IF SUPER^.Step(881, TRUE, 'Step number 881') THEN
    SUPER^.StepCompleteWhen((_runOneStep OR _runAllSteps) AND _finishStep);

    IF _runOneStep THEN
        _runOneStep := FALSE;
        RETURN;
    END_IF
END_IF

IF SUPER^.Step(882, TRUE, 'Step number 882') THEN
    SUPER^.StepCompleteWhen((_runOneStep OR _runAllSteps) AND _finishStep);

    IF _runOneStep THEN
        _runOneStep := FALSE;
        RETURN;
    END_IF
END_IF

IF SUPER^.Step(883, TRUE, 'Step number 883') THEN
    SUPER^.StepCompleteWhen((_runOneStep OR _runAllSteps) AND _finishStep);

    IF _runOneStep THEN
        _runOneStep := FALSE;
        RETURN;
    END_IF
END_IF

IF SUPER^.Step(884, TRUE, 'Step number 884') THEN
    SUPER^.StepCompleteWhen((_runOneStep OR _runAllSteps) AND _finishStep);

    IF _runOneStep THEN
        _runOneStep := FALSE;
        RETURN;
    END_IF
END_IF

IF SUPER^.Step(885, TRUE, 'Step number 885') THEN
    SUPER^.StepCompleteWhen((_runOneStep OR _runAllSteps) AND _finishStep);

    IF _runOneStep THEN
        _runOneStep := FALSE;
        RETURN;
    END_IF
END_IF

IF SUPER^.Step(886, TRUE, 'Step number 886') THEN
    SUPER^.StepCompleteWhen((_runOneStep OR _runAllSteps) AND _finishStep);

    IF _runOneStep THEN
        _runOneStep := FALSE;
        RETURN;
    END_IF
END_IF

IF SUPER^.Step(887, TRUE, 'Step number 887') THEN
    SUPER^.StepCompleteWhen((_runOneStep OR _runAllSteps) AND _finishStep);

    IF _runOneStep THEN
        _runOneStep := FALSE;
        RETURN;
    END_IF
END_IF

IF SUPER^.Step(888, TRUE, 'Step number 888') THEN
    SUPER^.StepCompleteWhen((_runOneStep OR _runAllSteps) AND _finishStep);

    IF _runOneStep THEN
        _runOneStep := FALSE;
        RETURN;
    END_IF
END_IF

IF SUPER^.Step(889, TRUE, 'Step number 889') THEN
    SUPER^.StepCompleteWhen((_runOneStep OR _runAllSteps) AND _finishStep);

    IF _runOneStep THEN
        _runOneStep := FALSE;
        RETURN;
    END_IF
END_IF

IF SUPER^.Step(890, TRUE, 'Step number 890') THEN
    SUPER^.StepCompleteWhen((_runOneStep OR _runAllSteps) AND _finishStep);

    IF _runOneStep THEN
        _runOneStep := FALSE;
        RETURN;
    END_IF
END_IF

IF SUPER^.Step(891, TRUE, 'Step number 891') THEN
    SUPER^.StepCompleteWhen((_runOneStep OR _runAllSteps) AND _finishStep);

    IF _runOneStep THEN
        _runOneStep := FALSE;
        RETURN;
    END_IF
END_IF

IF SUPER^.Step(892, TRUE, 'Step number 892') THEN
    SUPER^.StepCompleteWhen((_runOneStep OR _runAllSteps) AND _finishStep);

    IF _runOneStep THEN
        _runOneStep := FALSE;
        RETURN;
    END_IF
END_IF

IF SUPER^.Step(893, TRUE, 'Step number 893') THEN
    SUPER^.StepCompleteWhen((_runOneStep OR _runAllSteps) AND _finishStep);

    IF _runOneStep THEN
        _runOneStep := FALSE;
        RETURN;
    END_IF
END_IF

IF SUPER^.Step(894, TRUE, 'Step number 894') THEN
    SUPER^.StepCompleteWhen((_runOneStep OR _runAllSteps) AND _finishStep);

    IF _runOneStep THEN
        _runOneStep := FALSE;
        RETURN;
    END_IF
END_IF

IF SUPER^.Step(895, TRUE, 'Step number 895') THEN
    SUPER^.StepCompleteWhen((_runOneStep OR _runAllSteps) AND _finishStep);

    IF _runOneStep THEN
        _runOneStep := FALSE;
        RETURN;
    END_IF
END_IF

IF SUPER^.Step(896, TRUE, 'Step number 896') THEN
    SUPER^.StepCompleteWhen((_runOneStep OR _runAllSteps) AND _finishStep);

    IF _runOneStep THEN
        _runOneStep := FALSE;
        RETURN;
    END_IF
END_IF

IF SUPER^.Step(897, TRUE, 'Step number 897') THEN
    SUPER^.StepCompleteWhen((_runOneStep OR _runAllSteps) AND _finishStep);

    IF _runOneStep THEN
        _runOneStep := FALSE;
        RETURN;
    END_IF
END_IF

IF SUPER^.Step(898, TRUE, 'Step number 898') THEN
    SUPER^.StepCompleteWhen((_runOneStep OR _runAllSteps) AND _finishStep);

    IF _runOneStep THEN
        _runOneStep := FALSE;
        RETURN;
    END_IF
END_IF

IF SUPER^.Step(899, TRUE, 'Step number 899') THEN
    SUPER^.StepCompleteWhen((_runOneStep OR _runAllSteps) AND _finishStep);

    IF _runOneStep THEN
        _runOneStep := FALSE;
        RETURN;
    END_IF
END_IF

IF SUPER^.Step(900, TRUE, 'Step number 900') THEN
    SUPER^.StepCompleteWhen((_runOneStep OR _runAllSteps) AND _finishStep);

    IF _runOneStep THEN
        _runOneStep := FALSE;
        RETURN;
    END_IF
END_IF

IF SUPER^.Step(901, TRUE, 'Step number 901') THEN
    SUPER^.StepCompleteWhen((_runOneStep OR _runAllSteps) AND _finishStep);

    IF _runOneStep THEN
        _runOneStep := FALSE;
        RETURN;
    END_IF
END_IF

IF SUPER^.Step(902, TRUE, 'Step number 902') THEN
    SUPER^.StepCompleteWhen((_runOneStep OR _runAllSteps) AND _finishStep);

    IF _runOneStep THEN
        _runOneStep := FALSE;
        RETURN;
    END_IF
END_IF

IF SUPER^.Step(903, TRUE, 'Step number 903') THEN
    SUPER^.StepCompleteWhen((_runOneStep OR _runAllSteps) AND _finishStep);

    IF _runOneStep THEN
        _runOneStep := FALSE;
        RETURN;
    END_IF
END_IF

IF SUPER^.Step(904, TRUE, 'Step number 904') THEN
    SUPER^.StepCompleteWhen((_runOneStep OR _runAllSteps) AND _finishStep);

    IF _runOneStep THEN
        _runOneStep := FALSE;
        RETURN;
    END_IF
END_IF

IF SUPER^.Step(905, TRUE, 'Step number 905') THEN
    SUPER^.StepCompleteWhen((_runOneStep OR _runAllSteps) AND _finishStep);

    IF _runOneStep THEN
        _runOneStep := FALSE;
        RETURN;
    END_IF
END_IF

IF SUPER^.Step(906, TRUE, 'Step number 906') THEN
    SUPER^.StepCompleteWhen((_runOneStep OR _runAllSteps) AND _finishStep);

    IF _runOneStep THEN
        _runOneStep := FALSE;
        RETURN;
    END_IF
END_IF

IF SUPER^.Step(907, TRUE, 'Step number 907') THEN
    SUPER^.StepCompleteWhen((_runOneStep OR _runAllSteps) AND _finishStep);

    IF _runOneStep THEN
        _runOneStep := FALSE;
        RETURN;
    END_IF
END_IF

IF SUPER^.Step(908, TRUE, 'Step number 908') THEN
    SUPER^.StepCompleteWhen((_runOneStep OR _runAllSteps) AND _finishStep);

    IF _runOneStep THEN
        _runOneStep := FALSE;
        RETURN;
    END_IF
END_IF

IF SUPER^.Step(909, TRUE, 'Step number 909') THEN
    SUPER^.StepCompleteWhen((_runOneStep OR _runAllSteps) AND _finishStep);

    IF _runOneStep THEN
        _runOneStep := FALSE;
        RETURN;
    END_IF
END_IF

IF SUPER^.Step(910, TRUE, 'Step number 910') THEN
    SUPER^.StepCompleteWhen((_runOneStep OR _runAllSteps) AND _finishStep);

    IF _runOneStep THEN
        _runOneStep := FALSE;
        RETURN;
    END_IF
END_IF

IF SUPER^.Step(911, TRUE, 'Step number 911') THEN
    SUPER^.StepCompleteWhen((_runOneStep OR _runAllSteps) AND _finishStep);

    IF _runOneStep THEN
        _runOneStep := FALSE;
        RETURN;
    END_IF
END_IF

IF SUPER^.Step(912, TRUE, 'Step number 912') THEN
    SUPER^.StepCompleteWhen((_runOneStep OR _runAllSteps) AND _finishStep);

    IF _runOneStep THEN
        _runOneStep := FALSE;
        RETURN;
    END_IF
END_IF

IF SUPER^.Step(913, TRUE, 'Step number 913') THEN
    SUPER^.StepCompleteWhen((_runOneStep OR _runAllSteps) AND _finishStep);

    IF _runOneStep THEN
        _runOneStep := FALSE;
        RETURN;
    END_IF
END_IF

IF SUPER^.Step(914, TRUE, 'Step number 914') THEN
    SUPER^.StepCompleteWhen((_runOneStep OR _runAllSteps) AND _finishStep);

    IF _runOneStep THEN
        _runOneStep := FALSE;
        RETURN;
    END_IF
END_IF

IF SUPER^.Step(915, TRUE, 'Step number 915') THEN
    SUPER^.StepCompleteWhen((_runOneStep OR _runAllSteps) AND _finishStep);

    IF _runOneStep THEN
        _runOneStep := FALSE;
        RETURN;
    END_IF
END_IF

IF SUPER^.Step(916, TRUE, 'Step number 916') THEN
    SUPER^.StepCompleteWhen((_runOneStep OR _runAllSteps) AND _finishStep);

    IF _runOneStep THEN
        _runOneStep := FALSE;
        RETURN;
    END_IF
END_IF

IF SUPER^.Step(917, TRUE, 'Step number 917') THEN
    SUPER^.StepCompleteWhen((_runOneStep OR _runAllSteps) AND _finishStep);

    IF _runOneStep THEN
        _runOneStep := FALSE;
        RETURN;
    END_IF
END_IF

IF SUPER^.Step(918, TRUE, 'Step number 918') THEN
    SUPER^.StepCompleteWhen((_runOneStep OR _runAllSteps) AND _finishStep);

    IF _runOneStep THEN
        _runOneStep := FALSE;
        RETURN;
    END_IF
END_IF

IF SUPER^.Step(919, TRUE, 'Step number 919') THEN
    SUPER^.StepCompleteWhen((_runOneStep OR _runAllSteps) AND _finishStep);

    IF _runOneStep THEN
        _runOneStep := FALSE;
        RETURN;
    END_IF
END_IF

IF SUPER^.Step(920, TRUE, 'Step number 920') THEN
    SUPER^.StepCompleteWhen((_runOneStep OR _runAllSteps) AND _finishStep);

    IF _runOneStep THEN
        _runOneStep := FALSE;
        RETURN;
    END_IF
END_IF

IF SUPER^.Step(921, TRUE, 'Step number 921') THEN
    SUPER^.StepCompleteWhen((_runOneStep OR _runAllSteps) AND _finishStep);

    IF _runOneStep THEN
        _runOneStep := FALSE;
        RETURN;
    END_IF
END_IF

IF SUPER^.Step(922, TRUE, 'Step number 922') THEN
    SUPER^.StepCompleteWhen((_runOneStep OR _runAllSteps) AND _finishStep);

    IF _runOneStep THEN
        _runOneStep := FALSE;
        RETURN;
    END_IF
END_IF

IF SUPER^.Step(923, TRUE, 'Step number 923') THEN
    SUPER^.StepCompleteWhen((_runOneStep OR _runAllSteps) AND _finishStep);

    IF _runOneStep THEN
        _runOneStep := FALSE;
        RETURN;
    END_IF
END_IF

IF SUPER^.Step(924, TRUE, 'Step number 924') THEN
    SUPER^.StepCompleteWhen((_runOneStep OR _runAllSteps) AND _finishStep);

    IF _runOneStep THEN
        _runOneStep := FALSE;
        RETURN;
    END_IF
END_IF

IF SUPER^.Step(925, TRUE, 'Step number 925') THEN
    SUPER^.StepCompleteWhen((_runOneStep OR _runAllSteps) AND _finishStep);

    IF _runOneStep THEN
        _runOneStep := FALSE;
        RETURN;
    END_IF
END_IF

IF SUPER^.Step(926, TRUE, 'Step number 926') THEN
    SUPER^.StepCompleteWhen((_runOneStep OR _runAllSteps) AND _finishStep);

    IF _runOneStep THEN
        _runOneStep := FALSE;
        RETURN;
    END_IF
END_IF

IF SUPER^.Step(927, TRUE, 'Step number 927') THEN
    SUPER^.StepCompleteWhen((_runOneStep OR _runAllSteps) AND _finishStep);

    IF _runOneStep THEN
        _runOneStep := FALSE;
        RETURN;
    END_IF
END_IF

IF SUPER^.Step(928, TRUE, 'Step number 928') THEN
    SUPER^.StepCompleteWhen((_runOneStep OR _runAllSteps) AND _finishStep);

    IF _runOneStep THEN
        _runOneStep := FALSE;
        RETURN;
    END_IF
END_IF

IF SUPER^.Step(929, TRUE, 'Step number 929') THEN
    SUPER^.StepCompleteWhen((_runOneStep OR _runAllSteps) AND _finishStep);

    IF _runOneStep THEN
        _runOneStep := FALSE;
        RETURN;
    END_IF
END_IF

IF SUPER^.Step(930, TRUE, 'Step number 930') THEN
    SUPER^.StepCompleteWhen((_runOneStep OR _runAllSteps) AND _finishStep);

    IF _runOneStep THEN
        _runOneStep := FALSE;
        RETURN;
    END_IF
END_IF

IF SUPER^.Step(931, TRUE, 'Step number 931') THEN
    SUPER^.StepCompleteWhen((_runOneStep OR _runAllSteps) AND _finishStep);

    IF _runOneStep THEN
        _runOneStep := FALSE;
        RETURN;
    END_IF
END_IF

IF SUPER^.Step(932, TRUE, 'Step number 932') THEN
    SUPER^.StepCompleteWhen((_runOneStep OR _runAllSteps) AND _finishStep);

    IF _runOneStep THEN
        _runOneStep := FALSE;
        RETURN;
    END_IF
END_IF

IF SUPER^.Step(933, TRUE, 'Step number 933') THEN
    SUPER^.StepCompleteWhen((_runOneStep OR _runAllSteps) AND _finishStep);

    IF _runOneStep THEN
        _runOneStep := FALSE;
        RETURN;
    END_IF
END_IF

IF SUPER^.Step(934, TRUE, 'Step number 934') THEN
    SUPER^.StepCompleteWhen((_runOneStep OR _runAllSteps) AND _finishStep);

    IF _runOneStep THEN
        _runOneStep := FALSE;
        RETURN;
    END_IF
END_IF

IF SUPER^.Step(935, TRUE, 'Step number 935') THEN
    SUPER^.StepCompleteWhen((_runOneStep OR _runAllSteps) AND _finishStep);

    IF _runOneStep THEN
        _runOneStep := FALSE;
        RETURN;
    END_IF
END_IF

IF SUPER^.Step(936, TRUE, 'Step number 936') THEN
    SUPER^.StepCompleteWhen((_runOneStep OR _runAllSteps) AND _finishStep);

    IF _runOneStep THEN
        _runOneStep := FALSE;
        RETURN;
    END_IF
END_IF

IF SUPER^.Step(937, TRUE, 'Step number 937') THEN
    SUPER^.StepCompleteWhen((_runOneStep OR _runAllSteps) AND _finishStep);

    IF _runOneStep THEN
        _runOneStep := FALSE;
        RETURN;
    END_IF
END_IF

IF SUPER^.Step(938, TRUE, 'Step number 938') THEN
    SUPER^.StepCompleteWhen((_runOneStep OR _runAllSteps) AND _finishStep);

    IF _runOneStep THEN
        _runOneStep := FALSE;
        RETURN;
    END_IF
END_IF

IF SUPER^.Step(939, TRUE, 'Step number 939') THEN
    SUPER^.StepCompleteWhen((_runOneStep OR _runAllSteps) AND _finishStep);

    IF _runOneStep THEN
        _runOneStep := FALSE;
        RETURN;
    END_IF
END_IF

IF SUPER^.Step(940, TRUE, 'Step number 940') THEN
    SUPER^.StepCompleteWhen((_runOneStep OR _runAllSteps) AND _finishStep);

    IF _runOneStep THEN
        _runOneStep := FALSE;
        RETURN;
    END_IF
END_IF

IF SUPER^.Step(941, TRUE, 'Step number 941') THEN
    SUPER^.StepCompleteWhen((_runOneStep OR _runAllSteps) AND _finishStep);

    IF _runOneStep THEN
        _runOneStep := FALSE;
        RETURN;
    END_IF
END_IF

IF SUPER^.Step(942, TRUE, 'Step number 942') THEN
    SUPER^.StepCompleteWhen((_runOneStep OR _runAllSteps) AND _finishStep);

    IF _runOneStep THEN
        _runOneStep := FALSE;
        RETURN;
    END_IF
END_IF

IF SUPER^.Step(943, TRUE, 'Step number 943') THEN
    SUPER^.StepCompleteWhen((_runOneStep OR _runAllSteps) AND _finishStep);

    IF _runOneStep THEN
        _runOneStep := FALSE;
        RETURN;
    END_IF
END_IF

IF SUPER^.Step(944, TRUE, 'Step number 944') THEN
    SUPER^.StepCompleteWhen((_runOneStep OR _runAllSteps) AND _finishStep);

    IF _runOneStep THEN
        _runOneStep := FALSE;
        RETURN;
    END_IF
END_IF

IF SUPER^.Step(945, TRUE, 'Step number 945') THEN
    SUPER^.StepCompleteWhen((_runOneStep OR _runAllSteps) AND _finishStep);

    IF _runOneStep THEN
        _runOneStep := FALSE;
        RETURN;
    END_IF
END_IF

IF SUPER^.Step(946, TRUE, 'Step number 946') THEN
    SUPER^.StepCompleteWhen((_runOneStep OR _runAllSteps) AND _finishStep);

    IF _runOneStep THEN
        _runOneStep := FALSE;
        RETURN;
    END_IF
END_IF

IF SUPER^.Step(947, TRUE, 'Step number 947') THEN
    SUPER^.StepCompleteWhen((_runOneStep OR _runAllSteps) AND _finishStep);

    IF _runOneStep THEN
        _runOneStep := FALSE;
        RETURN;
    END_IF
END_IF

IF SUPER^.Step(948, TRUE, 'Step number 948') THEN
    SUPER^.StepCompleteWhen((_runOneStep OR _runAllSteps) AND _finishStep);

    IF _runOneStep THEN
        _runOneStep := FALSE;
        RETURN;
    END_IF
END_IF

IF SUPER^.Step(949, TRUE, 'Step number 949') THEN
    SUPER^.StepCompleteWhen((_runOneStep OR _runAllSteps) AND _finishStep);

    IF _runOneStep THEN
        _runOneStep := FALSE;
        RETURN;
    END_IF
END_IF

IF SUPER^.Step(950, TRUE, 'Step number 950') THEN
    SUPER^.StepCompleteWhen((_runOneStep OR _runAllSteps) AND _finishStep);

    IF _runOneStep THEN
        _runOneStep := FALSE;
        RETURN;
    END_IF
END_IF

IF SUPER^.Step(951, TRUE, 'Step number 951') THEN
    SUPER^.StepCompleteWhen((_runOneStep OR _runAllSteps) AND _finishStep);

    IF _runOneStep THEN
        _runOneStep := FALSE;
        RETURN;
    END_IF
END_IF

IF SUPER^.Step(952, TRUE, 'Step number 952') THEN
    SUPER^.StepCompleteWhen((_runOneStep OR _runAllSteps) AND _finishStep);

    IF _runOneStep THEN
        _runOneStep := FALSE;
        RETURN;
    END_IF
END_IF

IF SUPER^.Step(953, TRUE, 'Step number 953') THEN
    SUPER^.StepCompleteWhen((_runOneStep OR _runAllSteps) AND _finishStep);

    IF _runOneStep THEN
        _runOneStep := FALSE;
        RETURN;
    END_IF
END_IF

IF SUPER^.Step(954, TRUE, 'Step number 954') THEN
    SUPER^.StepCompleteWhen((_runOneStep OR _runAllSteps) AND _finishStep);

    IF _runOneStep THEN
        _runOneStep := FALSE;
        RETURN;
    END_IF
END_IF

IF SUPER^.Step(955, TRUE, 'Step number 955') THEN
    SUPER^.StepCompleteWhen((_runOneStep OR _runAllSteps) AND _finishStep);

    IF _runOneStep THEN
        _runOneStep := FALSE;
        RETURN;
    END_IF
END_IF

IF SUPER^.Step(956, TRUE, 'Step number 956') THEN
    SUPER^.StepCompleteWhen((_runOneStep OR _runAllSteps) AND _finishStep);

    IF _runOneStep THEN
        _runOneStep := FALSE;
        RETURN;
    END_IF
END_IF

IF SUPER^.Step(957, TRUE, 'Step number 957') THEN
    SUPER^.StepCompleteWhen((_runOneStep OR _runAllSteps) AND _finishStep);

    IF _runOneStep THEN
        _runOneStep := FALSE;
        RETURN;
    END_IF
END_IF

IF SUPER^.Step(958, TRUE, 'Step number 958') THEN
    SUPER^.StepCompleteWhen((_runOneStep OR _runAllSteps) AND _finishStep);

    IF _runOneStep THEN
        _runOneStep := FALSE;
        RETURN;
    END_IF
END_IF

IF SUPER^.Step(959, TRUE, 'Step number 959') THEN
    SUPER^.StepCompleteWhen((_runOneStep OR _runAllSteps) AND _finishStep);

    IF _runOneStep THEN
        _runOneStep := FALSE;
        RETURN;
    END_IF
END_IF

IF SUPER^.Step(960, TRUE, 'Step number 960') THEN
    SUPER^.StepCompleteWhen((_runOneStep OR _runAllSteps) AND _finishStep);

    IF _runOneStep THEN
        _runOneStep := FALSE;
        RETURN;
    END_IF
END_IF

IF SUPER^.Step(961, TRUE, 'Step number 961') THEN
    SUPER^.StepCompleteWhen((_runOneStep OR _runAllSteps) AND _finishStep);

    IF _runOneStep THEN
        _runOneStep := FALSE;
        RETURN;
    END_IF
END_IF

IF SUPER^.Step(962, TRUE, 'Step number 962') THEN
    SUPER^.StepCompleteWhen((_runOneStep OR _runAllSteps) AND _finishStep);

    IF _runOneStep THEN
        _runOneStep := FALSE;
        RETURN;
    END_IF
END_IF

IF SUPER^.Step(963, TRUE, 'Step number 963') THEN
    SUPER^.StepCompleteWhen((_runOneStep OR _runAllSteps) AND _finishStep);

    IF _runOneStep THEN
        _runOneStep := FALSE;
        RETURN;
    END_IF
END_IF

IF SUPER^.Step(964, TRUE, 'Step number 964') THEN
    SUPER^.StepCompleteWhen((_runOneStep OR _runAllSteps) AND _finishStep);

    IF _runOneStep THEN
        _runOneStep := FALSE;
        RETURN;
    END_IF
END_IF

IF SUPER^.Step(965, TRUE, 'Step number 965') THEN
    SUPER^.StepCompleteWhen((_runOneStep OR _runAllSteps) AND _finishStep);

    IF _runOneStep THEN
        _runOneStep := FALSE;
        RETURN;
    END_IF
END_IF

IF SUPER^.Step(966, TRUE, 'Step number 966') THEN
    SUPER^.StepCompleteWhen((_runOneStep OR _runAllSteps) AND _finishStep);

    IF _runOneStep THEN
        _runOneStep := FALSE;
        RETURN;
    END_IF
END_IF

IF SUPER^.Step(967, TRUE, 'Step number 967') THEN
    SUPER^.StepCompleteWhen((_runOneStep OR _runAllSteps) AND _finishStep);

    IF _runOneStep THEN
        _runOneStep := FALSE;
        RETURN;
    END_IF
END_IF

IF SUPER^.Step(968, TRUE, 'Step number 968') THEN
    SUPER^.StepCompleteWhen((_runOneStep OR _runAllSteps) AND _finishStep);

    IF _runOneStep THEN
        _runOneStep := FALSE;
        RETURN;
    END_IF
END_IF

IF SUPER^.Step(969, TRUE, 'Step number 969') THEN
    SUPER^.StepCompleteWhen((_runOneStep OR _runAllSteps) AND _finishStep);

    IF _runOneStep THEN
        _runOneStep := FALSE;
        RETURN;
    END_IF
END_IF

IF SUPER^.Step(970, TRUE, 'Step number 970') THEN
    SUPER^.StepCompleteWhen((_runOneStep OR _runAllSteps) AND _finishStep);

    IF _runOneStep THEN
        _runOneStep := FALSE;
        RETURN;
    END_IF
END_IF

IF SUPER^.Step(971, TRUE, 'Step number 971') THEN
    SUPER^.StepCompleteWhen((_runOneStep OR _runAllSteps) AND _finishStep);

    IF _runOneStep THEN
        _runOneStep := FALSE;
        RETURN;
    END_IF
END_IF

IF SUPER^.Step(972, TRUE, 'Step number 972') THEN
    SUPER^.StepCompleteWhen((_runOneStep OR _runAllSteps) AND _finishStep);

    IF _runOneStep THEN
        _runOneStep := FALSE;
        RETURN;
    END_IF
END_IF

IF SUPER^.Step(973, TRUE, 'Step number 973') THEN
    SUPER^.StepCompleteWhen((_runOneStep OR _runAllSteps) AND _finishStep);

    IF _runOneStep THEN
        _runOneStep := FALSE;
        RETURN;
    END_IF
END_IF

IF SUPER^.Step(974, TRUE, 'Step number 974') THEN
    SUPER^.StepCompleteWhen((_runOneStep OR _runAllSteps) AND _finishStep);

    IF _runOneStep THEN
        _runOneStep := FALSE;
        RETURN;
    END_IF
END_IF

IF SUPER^.Step(975, TRUE, 'Step number 975') THEN
    SUPER^.StepCompleteWhen((_runOneStep OR _runAllSteps) AND _finishStep);

    IF _runOneStep THEN
        _runOneStep := FALSE;
        RETURN;
    END_IF
END_IF

IF SUPER^.Step(976, TRUE, 'Step number 976') THEN
    SUPER^.StepCompleteWhen((_runOneStep OR _runAllSteps) AND _finishStep);

    IF _runOneStep THEN
        _runOneStep := FALSE;
        RETURN;
    END_IF
END_IF

IF SUPER^.Step(977, TRUE, 'Step number 977') THEN
    SUPER^.StepCompleteWhen((_runOneStep OR _runAllSteps) AND _finishStep);

    IF _runOneStep THEN
        _runOneStep := FALSE;
        RETURN;
    END_IF
END_IF

IF SUPER^.Step(978, TRUE, 'Step number 978') THEN
    SUPER^.StepCompleteWhen((_runOneStep OR _runAllSteps) AND _finishStep);

    IF _runOneStep THEN
        _runOneStep := FALSE;
        RETURN;
    END_IF
END_IF

IF SUPER^.Step(979, TRUE, 'Step number 979') THEN
    SUPER^.StepCompleteWhen((_runOneStep OR _runAllSteps) AND _finishStep);

    IF _runOneStep THEN
        _runOneStep := FALSE;
        RETURN;
    END_IF
END_IF

IF SUPER^.Step(980, TRUE, 'Step number 980') THEN
    SUPER^.StepCompleteWhen((_runOneStep OR _runAllSteps) AND _finishStep);

    IF _runOneStep THEN
        _runOneStep := FALSE;
        RETURN;
    END_IF
END_IF

IF SUPER^.Step(981, TRUE, 'Step number 981') THEN
    SUPER^.StepCompleteWhen((_runOneStep OR _runAllSteps) AND _finishStep);

    IF _runOneStep THEN
        _runOneStep := FALSE;
        RETURN;
    END_IF
END_IF

IF SUPER^.Step(982, TRUE, 'Step number 982') THEN
    SUPER^.StepCompleteWhen((_runOneStep OR _runAllSteps) AND _finishStep);

    IF _runOneStep THEN
        _runOneStep := FALSE;
        RETURN;
    END_IF
END_IF

IF SUPER^.Step(983, TRUE, 'Step number 983') THEN
    SUPER^.StepCompleteWhen((_runOneStep OR _runAllSteps) AND _finishStep);

    IF _runOneStep THEN
        _runOneStep := FALSE;
        RETURN;
    END_IF
END_IF

IF SUPER^.Step(984, TRUE, 'Step number 984') THEN
    SUPER^.StepCompleteWhen((_runOneStep OR _runAllSteps) AND _finishStep);

    IF _runOneStep THEN
        _runOneStep := FALSE;
        RETURN;
    END_IF
END_IF

IF SUPER^.Step(985, TRUE, 'Step number 985') THEN
    SUPER^.StepCompleteWhen((_runOneStep OR _runAllSteps) AND _finishStep);

    IF _runOneStep THEN
        _runOneStep := FALSE;
        RETURN;
    END_IF
END_IF

IF SUPER^.Step(986, TRUE, 'Step number 986') THEN
    SUPER^.StepCompleteWhen((_runOneStep OR _runAllSteps) AND _finishStep);

    IF _runOneStep THEN
        _runOneStep := FALSE;
        RETURN;
    END_IF
END_IF

IF SUPER^.Step(987, TRUE, 'Step number 987') THEN
    SUPER^.StepCompleteWhen((_runOneStep OR _runAllSteps) AND _finishStep);

    IF _runOneStep THEN
        _runOneStep := FALSE;
        RETURN;
    END_IF
END_IF

IF SUPER^.Step(988, TRUE, 'Step number 988') THEN
    SUPER^.StepCompleteWhen((_runOneStep OR _runAllSteps) AND _finishStep);

    IF _runOneStep THEN
        _runOneStep := FALSE;
        RETURN;
    END_IF
END_IF

IF SUPER^.Step(989, TRUE, 'Step number 989') THEN
    SUPER^.StepCompleteWhen((_runOneStep OR _runAllSteps) AND _finishStep);

    IF _runOneStep THEN
        _runOneStep := FALSE;
        RETURN;
    END_IF
END_IF

IF SUPER^.Step(990, TRUE, 'Step number 990') THEN
    SUPER^.StepCompleteWhen((_runOneStep OR _runAllSteps) AND _finishStep);

    IF _runOneStep THEN
        _runOneStep := FALSE;
        RETURN;
    END_IF
END_IF

IF SUPER^.Step(991, TRUE, 'Step number 991') THEN
    SUPER^.StepCompleteWhen((_runOneStep OR _runAllSteps) AND _finishStep);

    IF _runOneStep THEN
        _runOneStep := FALSE;
        RETURN;
    END_IF
END_IF

IF SUPER^.Step(992, TRUE, 'Step number 992') THEN
    SUPER^.StepCompleteWhen((_runOneStep OR _runAllSteps) AND _finishStep);

    IF _runOneStep THEN
        _runOneStep := FALSE;
        RETURN;
    END_IF
END_IF

IF SUPER^.Step(993, TRUE, 'Step number 993') THEN
    SUPER^.StepCompleteWhen((_runOneStep OR _runAllSteps) AND _finishStep);

    IF _runOneStep THEN
        _runOneStep := FALSE;
        RETURN;
    END_IF
END_IF

IF SUPER^.Step(994, TRUE, 'Step number 994') THEN
    SUPER^.StepCompleteWhen((_runOneStep OR _runAllSteps) AND _finishStep);

    IF _runOneStep THEN
        _runOneStep := FALSE;
        RETURN;
    END_IF
END_IF

IF SUPER^.Step(995, TRUE, 'Step number 995') THEN
    SUPER^.StepCompleteWhen((_runOneStep OR _runAllSteps) AND _finishStep);

    IF _runOneStep THEN
        _runOneStep := FALSE;
        RETURN;
    END_IF
END_IF

IF SUPER^.Step(996, TRUE, 'Step number 996') THEN
    SUPER^.StepCompleteWhen((_runOneStep OR _runAllSteps) AND _finishStep);

    IF _runOneStep THEN
        _runOneStep := FALSE;
        RETURN;
    END_IF
END_IF

IF SUPER^.Step(997, TRUE, 'Step number 997') THEN
    SUPER^.StepCompleteWhen((_runOneStep OR _runAllSteps) AND _finishStep);

    IF _runOneStep THEN
        _runOneStep := FALSE;
        RETURN;
    END_IF
END_IF

IF SUPER^.Step(998, TRUE, 'Step number 998') THEN
    SUPER^.StepCompleteWhen((_runOneStep OR _runAllSteps) AND _finishStep);

    IF _runOneStep THEN
        _runOneStep := FALSE;
        RETURN;
    END_IF
END_IF

IF SUPER^.Step(999, TRUE, 'Step number 999') THEN
    SUPER^.StepCompleteWhen((_runOneStep OR _runAllSteps) AND _finishStep);

    IF _runOneStep THEN
        _runOneStep := FALSE;
        RETURN;
    END_IF
END_IF

IF SUPER^.Step(1000, TRUE, 'Step number 1000') THEN
    SUPER^.StepCompleteWhen((_runOneStep OR _runAllSteps) AND _finishStep);

    IF _runOneStep THEN
        _runOneStep := FALSE;
        RETURN;
    END_IF
END_IF

IF SUPER^.Step(1001, TRUE, 'Step number 1001') THEN
    SUPER^.StepCompleteWhen((_runOneStep OR _runAllSteps) AND _finishStep);

    IF _runOneStep THEN
        _runOneStep := FALSE;
        RETURN;
    END_IF
END_IF

IF SUPER^.Step(1002, TRUE, 'Step number 1002') THEN
    SUPER^.StepCompleteWhen((_runOneStep OR _runAllSteps) AND _finishStep);

    IF _runOneStep THEN
        _runOneStep := FALSE;
        RETURN;
    END_IF
END_IF

IF SUPER^.Step(1003, TRUE, 'Step number 1003') THEN
    SUPER^.StepCompleteWhen((_runOneStep OR _runAllSteps) AND _finishStep);

    IF _runOneStep THEN
        _runOneStep := FALSE;
        RETURN;
    END_IF
END_IF

IF SUPER^.Step(1004, TRUE, 'Step number 1004') THEN
    SUPER^.StepCompleteWhen((_runOneStep OR _runAllSteps) AND _finishStep);

    IF _runOneStep THEN
        _runOneStep := FALSE;
        RETURN;
    END_IF
END_IF

IF SUPER^.Step(1005, TRUE, 'Step number 1005') THEN
    SUPER^.StepCompleteWhen((_runOneStep OR _runAllSteps) AND _finishStep);

    IF _runOneStep THEN
        _runOneStep := FALSE;
        RETURN;
    END_IF
END_IF

IF SUPER^.Step(1006, TRUE, 'Step number 1006') THEN
    SUPER^.StepCompleteWhen((_runOneStep OR _runAllSteps) AND _finishStep);

    IF _runOneStep THEN
        _runOneStep := FALSE;
        RETURN;
    END_IF
END_IF

IF SUPER^.Step(1007, TRUE, 'Step number 1007') THEN
    SUPER^.StepCompleteWhen((_runOneStep OR _runAllSteps) AND _finishStep);

    IF _runOneStep THEN
        _runOneStep := FALSE;
        RETURN;
    END_IF
END_IF

IF SUPER^.Step(1008, TRUE, 'Step number 1008') THEN
    SUPER^.StepCompleteWhen((_runOneStep OR _runAllSteps) AND _finishStep);

    IF _runOneStep THEN
        _runOneStep := FALSE;
        RETURN;
    END_IF
END_IF

IF SUPER^.Step(1009, TRUE, 'Step number 1009') THEN
    SUPER^.StepCompleteWhen((_runOneStep OR _runAllSteps) AND _finishStep);

    IF _runOneStep THEN
        _runOneStep := FALSE;
        RETURN;
    END_IF
END_IF

IF SUPER^.Step(1010, TRUE, 'Step number 1010') THEN
    SUPER^.StepCompleteWhen((_runOneStep OR _runAllSteps) AND _finishStep);

    IF _runOneStep THEN
        _runOneStep := FALSE;
        RETURN;
    END_IF
END_IF

IF SUPER^.Step(1011, TRUE, 'Step number 1011') THEN
    SUPER^.StepCompleteWhen((_runOneStep OR _runAllSteps) AND _finishStep);

    IF _runOneStep THEN
        _runOneStep := FALSE;
        RETURN;
    END_IF
END_IF

IF SUPER^.Step(1012, TRUE, 'Step number 1012') THEN
    SUPER^.StepCompleteWhen((_runOneStep OR _runAllSteps) AND _finishStep);

    IF _runOneStep THEN
        _runOneStep := FALSE;
        RETURN;
    END_IF
END_IF

IF SUPER^.Step(1013, TRUE, 'Step number 1013') THEN
    SUPER^.StepCompleteWhen((_runOneStep OR _runAllSteps) AND _finishStep);

    IF _runOneStep THEN
        _runOneStep := FALSE;
        RETURN;
    END_IF
END_IF

IF SUPER^.Step(1014, TRUE, 'Step number 1014') THEN
    SUPER^.StepCompleteWhen((_runOneStep OR _runAllSteps) AND _finishStep);

    IF _runOneStep THEN
        _runOneStep := FALSE;
        RETURN;
    END_IF
END_IF

IF SUPER^.Step(1015, TRUE, 'Step number 1015') THEN
    SUPER^.StepCompleteWhen((_runOneStep OR _runAllSteps) AND _finishStep);

    IF _runOneStep THEN
        _runOneStep := FALSE;
        RETURN;
    END_IF
END_IF

IF SUPER^.Step(1016, TRUE, 'Step number 1016') THEN
    SUPER^.StepCompleteWhen((_runOneStep OR _runAllSteps) AND _finishStep);

    IF _runOneStep THEN
        _runOneStep := FALSE;
        RETURN;
    END_IF
END_IF

IF SUPER^.Step(1017, TRUE, 'Step number 1017') THEN
    SUPER^.StepCompleteWhen((_runOneStep OR _runAllSteps) AND _finishStep);

    IF _runOneStep THEN
        _runOneStep := FALSE;
        RETURN;
    END_IF
END_IF

IF SUPER^.Step(1018, TRUE, 'Step number 1018') THEN
    SUPER^.StepCompleteWhen((_runOneStep OR _runAllSteps) AND _finishStep);

    IF _runOneStep THEN
        _runOneStep := FALSE;
        RETURN;
    END_IF
END_IF

IF SUPER^.Step(1019, TRUE, 'Step number 1019') THEN
    SUPER^.StepCompleteWhen((_runOneStep OR _runAllSteps) AND _finishStep);

    IF _runOneStep THEN
        _runOneStep := FALSE;
        RETURN;
    END_IF
END_IF

IF SUPER^.Step(1020, TRUE, 'Step number 1020') THEN
    SUPER^.StepCompleteWhen((_runOneStep OR _runAllSteps) AND _finishStep);

    IF _runOneStep THEN
        _runOneStep := FALSE;
        RETURN;
    END_IF
END_IF

IF SUPER^.Step(1021, TRUE, 'Step number 1021') THEN
    SUPER^.StepCompleteWhen((_runOneStep OR _runAllSteps) AND _finishStep);

    IF _runOneStep THEN
        _runOneStep := FALSE;
        RETURN;
    END_IF
END_IF

IF SUPER^.Step(1022, TRUE, 'Step number 1022') THEN
    SUPER^.StepCompleteWhen((_runOneStep OR _runAllSteps) AND _finishStep);

    IF _runOneStep THEN
        _runOneStep := FALSE;
        RETURN;
    END_IF
END_IF

IF SUPER^.Step(1023, TRUE, 'Step number 1023') THEN
    SUPER^.StepCompleteWhen((_runOneStep OR _runAllSteps) AND _finishStep);

    IF _runOneStep THEN
        _runOneStep := FALSE;
        RETURN;
    END_IF
END_IF

//******************************************************************
IF SUPER^.Step(_stepId, _enabled, _stepDescription) THEN
    SUPER^.StepCompleteWhen((_runOneStep OR _runAllSteps) AND _finishStep);

    IF _runOneStep THEN
        _runOneStep := FALSE;
        RETURN;
    END_IF
END_IF
END_METHOD

METHOD MAIN_CommentOutPartOfRunningSequencer
VAR
    i : INT;
END_VAR
IF _sequenceRun = 1 THEN
    IF Step(0, TRUE, 'Step 0') THEN
        StepCompleteWhen(TRUE);
    END_IF

    IF Step(1, TRUE, 'Step 1') THEN
        StepCompleteWhen(TRUE);
    END_IF

    IF Step(2, TRUE, 'Step 2') THEN
        StepCompleteWhen(TRUE);
    END_IF

    IF Step(3, TRUE, 'Step 3') THEN
        StepCompleteWhen(FALSE);
    END_IF

    FOR i := 4 TO _totalStepNumber - 2 DO
        IF Step(i, TRUE, CONCAT('Step ', INT_TO_STRING(i))) THEN
            StepCompleteWhen(FALSE);
        END_IF
    END_FOR

    IF Step(_totalStepNumber - 1, TRUE, CONCAT('Step ', INT_TO_STRING(_totalStepNumber - 1))) THEN
        _SequenceComplete();
    END_IF
END_IF

IF _sequenceRun >= 2 THEN
    IF Step(0, TRUE, 'Step 0') THEN
        StepCompleteWhen(TRUE);
    END_IF

    //	IF Step(1, TRUE, 'Step 1') THEN
    //	   StepCompleteWhen(TRUE);
    //	END_IF
    //	IF Step(2, TRUE, 'Step 2') THEN
    //	   StepCompleteWhen(TRUE);
    //	END_IF
    IF Step(3, TRUE, 'Step 3') THEN
        StepCompleteWhen(FALSE);
    END_IF

    FOR i := 4 TO _totalStepNumber - 2 DO
        IF Step(i, TRUE, CONCAT('Step ', INT_TO_STRING(i))) THEN
            StepCompleteWhen(FALSE);
        END_IF
    END_FOR

    IF Step(_totalStepNumber - 1, TRUE, CONCAT('Step ', INT_TO_STRING(_totalStepNumber - 1))) THEN
        _SequenceComplete();
    END_IF
END_IF
END_METHOD

METHOD MAIN_ExecutionInOnePLCcycle
VAR
    i : INT;
END_VAR
FOR i := 0 TO _totalStepNumber - 2 DO
    IF Step(i, TRUE, CONCAT('Step ', INT_TO_STRING(i))) THEN
        StepCompleteWhen(TRUE);
    END_IF
END_FOR

IF Step(_totalStepNumber - 1, TRUE, CONCAT('Step ', INT_TO_STRING(_totalStepNumber - 1))) THEN
    _SequenceComplete();
END_IF
END_METHOD

METHOD MAIN_MaxStepId
VAR
    i : INT;
END_VAR
FOR i := 0 TO _totalStepNumber - 1 DO
    IF Step(i, TRUE, CONCAT('Step ', INT_TO_STRING(i))) THEN
        StepCompleteWhen(_finishStep);
    END_IF
END_FOR

IF Step(_stepId, TRUE, CONCAT('Step ', INT_TO_STRING(_stepId))) THEN
    StepCompleteWhen(TRUE);
END_IF
END_METHOD

METHOD MAIN_MinStepId
VAR
    i : INT;
END_VAR
IF Step(_stepId, TRUE, CONCAT('Step ', INT_TO_STRING(_stepId))) THEN
    StepCompleteWhen(TRUE);
END_IF

FOR i := 1 TO _totalStepNumber - 1 DO
    IF Step(i, TRUE, CONCAT('Step ', INT_TO_STRING(i))) THEN
        StepCompleteWhen(_finishStep);
    END_IF
END_FOR
END_METHOD

METHOD MAIN_NumberOfStepsCount
VAR
    i : INT;
END_VAR
IF Step(0, TRUE, 'Step 0') THEN
    StepCompleteWhen(TRUE);
END_IF

FOR i := 1 TO _totalStepNumber - 1 DO
    IF Step(i, TRUE, CONCAT('Step ', INT_TO_STRING(i))) THEN
        StepCompleteWhen(_finishStep);
    END_IF
END_FOR
END_METHOD

METHOD MAIN_OnStateChangeWhenChangingModes
VAR
    i : INT;
END_VAR
IF _sequenceRun <= _cyclicCycles OR _sequenceRun > _cyclicCycles + _stepInEvents + 1 THEN
    SetCyclicMode();

    FOR i := 0 TO _totalStepNumber - 2 DO
        IF Step(i, TRUE, CONCAT('Step ', INT_TO_STRING(i))) THEN
            _StepCompleteWhen(TRUE);
        END_IF
    END_FOR

    IF Step(_totalStepNumber - 1, TRUE, CONCAT('Step ', INT_TO_STRING(_totalStepNumber - 1))) THEN
        CompleteSequence();
        _sequenceCycles := _sequenceCycles + 1;
    END_IF
END_IF

IF _sequenceRun = _cyclicCycles + 1 THEN
    SetStepMode();
    Step(0, FALSE, '');
END_IF

IF _sequenceRun > _cyclicCycles + 1 AND _sequenceRun <= _cyclicCycles + _stepInEvents + 1 THEN
    SetStepMode();
    _StepIn();

    FOR i := 0 TO _totalStepNumber - 2 DO
        IF Step(i, TRUE, CONCAT('Step ', INT_TO_STRING(i))) THEN
            _StepCompleteWhen(TRUE);
        END_IF
    END_FOR

    IF Step(_totalStepNumber - 1, TRUE, CONCAT('Step ', INT_TO_STRING(_totalStepNumber - 1))) THEN
        CompleteSequence();
        _sequenceCycles := _sequenceCycles + 1;
    END_IF
END_IF
END_METHOD

METHOD MAIN_RequestStep
VAR
    i : INT;
END_VAR
IF _sequenceRun = 1 THEN
    FOR i := -5 TO -1 DO
        IF Step(i, TRUE, CONCAT('Step ', INT_TO_STRING(i))) THEN
            StepCompleteWhen(TRUE);
        END_IF
    END_FOR

    IF Step(0, TRUE, 'Step 0') THEN
        RequestStep(-5);
    END_IF

    FOR i := 1 TO 5 DO
        IF Step(i, TRUE, CONCAT('Step ', INT_TO_STRING(i))) THEN
            StepCompleteWhen(TRUE);
        END_IF
    END_FOR
END_IF

IF _sequenceRun = 2 THEN
    FOR i := -5 TO 5 DO
        IF Step(i, TRUE, CONCAT('Step ', INT_TO_STRING(i))) THEN
            StepCompleteWhen(FALSE);
        END_IF
    END_FOR
END_IF

IF _sequenceRun = 3 THEN
    IF Step(-5, TRUE, 'Step -5') THEN
        RequestStep(0);
    END_IF

    FOR i := -4 TO 5 DO
        IF Step(i, TRUE, CONCAT('Step ', INT_TO_STRING(i))) THEN
            StepCompleteWhen(FALSE);
        END_IF
    END_FOR
END_IF
END_METHOD

METHOD MAIN_RequestStepFromHigherToLower
VAR
    i : INT;
END_VAR
IF _sequenceRun = 1 THEN
    FOR i := 0 TO _reqStep + 4 DO
        IF Step(i, TRUE, CONCAT('Step ', INT_TO_STRING(i))) THEN
            StepCompleteWhen(TRUE);
        END_IF
    END_FOR

    FOR i := _reqStep + 5 TO _totalStepNumber - 2 DO
        Step(i, TRUE, CONCAT('Step ', INT_TO_STRING(i)));
    END_FOR

    RequestStep(_reqStep);

    IF Step(_totalStepNumber - 1, TRUE, CONCAT('Step ', INT_TO_STRING(_totalStepNumber - 1))) THEN
        _SequenceComplete();
    END_IF
END_IF

IF _sequenceRun = 2 THEN
    FOR i := 0 TO _totalStepNumber - 2 DO
        Step(i, TRUE, CONCAT('Step ', INT_TO_STRING(i)));
    END_FOR

    IF Step(_totalStepNumber - 1, TRUE, CONCAT('Step ', INT_TO_STRING(_totalStepNumber - 1))) THEN
        _SequenceComplete();
    END_IF
END_IF
END_METHOD

METHOD MAIN_RequestStepFromLowerToHigher
VAR
    i : INT;
END_VAR
IF _sequenceRun = 1 THEN
    IF Step(0, TRUE, 'Step 0') THEN
        StepCompleteWhen(TRUE);
    END_IF

    FOR i := 1 TO _totalStepNumber - 2 DO
        Step(i, TRUE, CONCAT('Step ', INT_TO_STRING(i)));
    END_FOR

    IF Step(_totalStepNumber - 1, TRUE, CONCAT('Step ', INT_TO_STRING(_totalStepNumber - 1))) THEN
        _SequenceComplete();
    END_IF
END_IF

IF _sequenceRun = 2 THEN
    IF Step(0, TRUE, 'Step 0') THEN
        StepCompleteWhen(TRUE);
    END_IF

    RequestStep(_reqStep);

    FOR i := 1 TO _totalStepNumber - 2 DO
        Step(i, TRUE, CONCAT('Step ', INT_TO_STRING(i)));
    END_FOR

    IF Step(_totalStepNumber - 1, TRUE, CONCAT('Step ', INT_TO_STRING(_totalStepNumber - 1))) THEN
        _SequenceComplete();
    END_IF
END_IF
END_METHOD

METHOD MAIN_RequestStepToFirstStepWithStepId0
VAR
    i : INT;
END_VAR
FOR i := 0 TO 4 DO
    IF Step(i, TRUE, CONCAT('Step ', INT_TO_STRING(i))) THEN
        StepCompleteWhen(_finishStep);
    END_IF
END_FOR

IF Step(5, TRUE, 'Step 5') THEN
    RequestStep(0);
END_IF

FOR i := 6 TO _totalStepNumber - 1 DO
    IF Step(i, TRUE, CONCAT('Step ', INT_TO_STRING(i))) THEN
        StepCompleteWhen(_finishStep);
    END_IF
END_FOR
END_METHOD

METHOD MAIN_RequestStepToNotExistingStep
VAR
    i : INT;
END_VAR
IF _sequenceRun = 1 THEN
    RequestStep(_reqStepNotExists);

    FOR i := 0 TO _totalStepNumber - 2 DO
        Step(i, TRUE, CONCAT('Step ', INT_TO_STRING(i)));
    END_FOR

    IF Step(_totalStepNumber - 1, TRUE, CONCAT('Step ', INT_TO_STRING(_totalStepNumber - 1))) THEN
        _SequenceComplete();
    END_IF
END_IF

IF _sequenceRun >= 2 THEN
    FOR i := 0 TO _totalStepNumber - 2 DO
        Step(i, TRUE, CONCAT('Step ', INT_TO_STRING(i)));
    END_FOR

    IF Step(_totalStepNumber - 1, TRUE, CONCAT('Step ', INT_TO_STRING(_totalStepNumber - 1))) THEN
        _SequenceComplete();
    END_IF
END_IF
END_METHOD

METHOD MAIN_RequestStepWhilePreviousRequestStepHasNotBeenYetProcessed
VAR
    i : INT;
END_VAR
FOR i := 0 TO _reqStep + 4 DO
    IF Step(i, TRUE, CONCAT('Step ', INT_TO_STRING(i))) THEN
        StepCompleteWhen(TRUE);
    END_IF
END_FOR

RequestStep(_reqStep);

FOR i := _reqStep + 5 TO _totalStepNumber - 2 DO
    Step(i, TRUE, CONCAT('Step ', INT_TO_STRING(i)));
END_FOR

RequestStep(_reqStep + 10);

IF Step(_totalStepNumber - 1, TRUE, CONCAT('Step ', INT_TO_STRING(_totalStepNumber - 1))) THEN
    _SequenceComplete();
END_IF
END_METHOD

METHOD MAIN_RestoreChildBetweenSteps
VAR
    i : INT;
    _childState : INT;
END_VAR
FOR i := 0 TO _totalStepNumber - 2 DO
    IF Step(i, TRUE, CONCAT('Step ', INT_TO_STRING(i))) THEN
        _childState := _myTcoChildState.State;
        _myTcoChildState.ChangeState(_myTcoChildState._requestedState);
        StepCompleteWhen(TRUE);
    END_IF
END_FOR

IF Step(_totalStepNumber - 1, TRUE, CONCAT('Step ', INT_TO_STRING(_totalStepNumber - 1))) THEN
    _SequenceComplete();
END_IF
END_METHOD

METHOD MAIN_SetStepMode
VAR
    i : INT;
END_VAR
IF _sequenceRun = 1 THEN
    IF Step(0, TRUE, 'Initial step') THEN
        StepCompleteWhen(TRUE);
    END_IF

    FOR i := 1 TO _totalStepNumber - 2 DO
        Step(i, TRUE, CONCAT('Step ', INT_TO_STRING(i)));
    END_FOR

    IF Step(_totalStepNumber - 1, TRUE, CONCAT('Step ', INT_TO_STRING(_totalStepNumber - 1))) THEN
        _SequenceComplete();
    END_IF
END_IF

IF _sequenceRun = 4 THEN
    IF Step(0, TRUE, 'Initial step') THEN
        StepCompleteWhen(TRUE);
    END_IF

    FOR i := 1 TO _totalStepNumber - 2 DO
        IF Step(i, TRUE, CONCAT('Step ', INT_TO_STRING(i))) THEN
            StepCompleteWhen(TRUE);
        END_IF
    END_FOR

    IF Step(_totalStepNumber - 1, TRUE, CONCAT('Step ', INT_TO_STRING(_totalStepNumber - 1))) THEN
        _SequenceComplete();
    END_IF
END_IF
END_METHOD

METHOD MAIN_StepMode
VAR
    i : INT;
END_VAR
IF _sequenceRun = 1 THEN
    IF Step(0, TRUE, 'Initial step') THEN
        StepCompleteWhen(TRUE);
    END_IF

    FOR i := 1 TO _totalStepNumber - 2 DO
        Step(i, TRUE, CONCAT('Step ', INT_TO_STRING(i)));
    END_FOR

    IF Step(_totalStepNumber - 1, TRUE, CONCAT('Step ', INT_TO_STRING(_totalStepNumber - 1))) THEN
        _SequenceComplete();
    END_IF
END_IF

IF _sequenceRun > 1 THEN
    _StepIn();

    IF Step(0, TRUE, 'Initial step') THEN
        StepCompleteWhen(TRUE);
    END_IF

    FOR i := 1 TO _totalStepNumber - 2 DO
        IF Step(i, TRUE, CONCAT('Step ', INT_TO_STRING(i))) THEN
            StepCompleteWhen(TRUE);
        END_IF
    END_FOR

    IF Step(_totalStepNumber - 1, TRUE, CONCAT('Step ', INT_TO_STRING(_totalStepNumber - 1))) THEN
        _SequenceComplete();
    END_IF
END_IF
END_METHOD

METHOD MAIN_StepModeChangeStepIdDuringExecution
VAR
    i : INT;
END_VAR
IF _sequenceRun = 1 THEN
    IF _currentStep.Status = 20 THEN
        _StepIn();
    END_IF

    // Step 0
    IF Step(0, TRUE, 'Step 0') THEN
        StepCompleteWhen(TRUE);
    END_IF

    // Step 1
    IF Step(1, TRUE, 'Step 1') THEN
        StepCompleteWhen(TRUE);
    END_IF

    // Step 2
    IF Step(2, TRUE, 'Step 2') THEN
        StepCompleteWhen(TRUE);
    END_IF

    // Step 3
    IF Step(3, TRUE, 'Step 3') THEN
        StepCompleteWhen(FALSE);
    END_IF

    FOR i := 4 TO _totalStepNumber - 2 DO
        Step(i, TRUE, CONCAT('Step  ', INT_TO_STRING(i)));
    END_FOR

    IF Step(_totalStepNumber - 1, TRUE, CONCAT('Step  ', INT_TO_STRING(_totalStepNumber - 1))) THEN
        _SequenceComplete();
    END_IF
END_IF

IF _sequenceRun = 2 THEN
    IF _currentStep.Status = 20 THEN
        _StepIn();
    END_IF

    // Step 0
    IF Step(0, TRUE, 'Step 0') THEN
        StepCompleteWhen(TRUE);
    END_IF

    // Step 1
    IF Step(1, TRUE, 'Step 1') THEN
        StepCompleteWhen(TRUE);
    END_IF

    // Step 2
    IF Step(2, TRUE, 'Step 2') THEN
        StepCompleteWhen(TRUE);
    END_IF

    // Step 3
    IF Step(5, TRUE, 'Step 3') THEN
        StepCompleteWhen(FALSE);
    END_IF

    FOR i := 4 TO _totalStepNumber - 2 DO
        Step(i, TRUE, CONCAT('Step  ', INT_TO_STRING(i)));
    END_FOR

    IF Step(_totalStepNumber - 1, TRUE, CONCAT('Step  ', INT_TO_STRING(_totalStepNumber - 1))) THEN
        _SequenceComplete();
    END_IF
END_IF
END_METHOD

METHOD MAIN_StepModeChangeStepOrder
VAR
    i : INT;
END_VAR
IF _sequenceRun <= _totalStepNumber + 1 THEN
    IF _currentStep.Status = 20 THEN
        _StepIn();
    END_IF

    // Step 0
    IF Step(0, TRUE, 'Step 0') THEN
        StepCompleteWhen(TRUE);
    END_IF

    // Step 1
    IF Step(1, TRUE, 'Step 1') THEN
        StepCompleteWhen(TRUE);
    END_IF

    // Step 2
    IF Step(2, TRUE, 'Step 2') THEN
        StepCompleteWhen(TRUE);
    END_IF

    // Step 3
    IF Step(3, TRUE, 'Step 3') THEN
        StepCompleteWhen(FALSE);
    END_IF

    FOR i := 4 TO _totalStepNumber - 2 DO
        Step(i, TRUE, CONCAT('Step  ', INT_TO_STRING(i)));
    END_FOR

    IF Step(_totalStepNumber - 1, TRUE, CONCAT('Step  ', INT_TO_STRING(_totalStepNumber - 1))) THEN
        _SequenceComplete();
    END_IF
END_IF

IF _sequenceRun = _totalStepNumber + 2 THEN
    IF _currentStep.Status = 20 THEN
        _StepIn();
    END_IF

    // Step 0
    IF Step(0, TRUE, 'Step 0') THEN
        StepCompleteWhen(TRUE);
    END_IF

    // Step 1
    IF Step(1, TRUE, 'Step 1') THEN
        StepCompleteWhen(TRUE);
    END_IF

    // Step 3
    IF Step(3, TRUE, 'Step 3') THEN
        StepCompleteWhen(FALSE);
    END_IF

    // Step 2
    IF Step(2, TRUE, 'Step 2') THEN
        StepCompleteWhen(TRUE);
    END_IF

    FOR i := 4 TO _totalStepNumber - 2 DO
        Step(i, TRUE, CONCAT('Step  ', INT_TO_STRING(i)));
    END_FOR

    IF Step(_totalStepNumber - 1, TRUE, CONCAT('Step  ', INT_TO_STRING(_totalStepNumber - 1))) THEN
        _SequenceComplete();
    END_IF
END_IF
END_METHOD

METHOD MAIN_StepModeCommentOutPartOfRunningSequencer
VAR
    i : INT;
END_VAR
IF _sequenceRun = 1 THEN
    IF (_currentStep.Status = 20) THEN
        _StepIn();
    END_IF

    IF Step(0, TRUE, 'Step 0') THEN
        StepCompleteWhen(TRUE);
    END_IF

    IF Step(1, TRUE, 'Step 1') THEN
        StepCompleteWhen(TRUE);
    END_IF

    IF Step(2, TRUE, 'Step 2') THEN
        StepCompleteWhen(TRUE);
    END_IF

    IF Step(3, TRUE, 'Step 3') THEN
        StepCompleteWhen(FALSE);
    END_IF

    FOR i := 4 TO _totalStepNumber - 2 DO
        IF Step(i, TRUE, CONCAT('Step ', INT_TO_STRING(i))) THEN
            StepCompleteWhen(FALSE);
        END_IF
    END_FOR

    IF Step(_totalStepNumber - 1, TRUE, CONCAT('Step ', INT_TO_STRING(_totalStepNumber - 1))) THEN
        _SequenceComplete();
    END_IF
END_IF

IF _sequenceRun >= 2 THEN
    IF (_currentStep.Status = 20) THEN
        _StepIn();
    END_IF

    IF Step(0, TRUE, 'Step 0') THEN
        StepCompleteWhen(TRUE);
    END_IF

    //	IF Step(1, TRUE, 'Step 1') THEN
    //	   StepCompleteWhen(TRUE);
    //	END_IF
    //	IF Step(2, TRUE, 'Step 2') THEN
    //	   StepCompleteWhen(TRUE);
    //	END_IF
    IF Step(3, TRUE, 'Step 3') THEN
        StepCompleteWhen(FALSE);
    END_IF

    FOR i := 4 TO _totalStepNumber - 2 DO
        IF Step(i, TRUE, CONCAT('Step ', INT_TO_STRING(i))) THEN
            StepCompleteWhen(FALSE);
        END_IF
    END_FOR

    IF Step(_totalStepNumber - 1, TRUE, CONCAT('Step ', INT_TO_STRING(_totalStepNumber - 1))) THEN
        _SequenceComplete();
    END_IF
END_IF
END_METHOD

METHOD MAIN_StepModeDisabledStep
VAR
    i : INT;
END_VAR
IF _sequenceRun = 1 THEN
    FOR i := 0 TO _totalStepNumber - 1 DO
        Step(i, TRUE, CONCAT('Step ', INT_TO_STRING(i)));
    END_FOR
END_IF

IF _sequenceRun = 2 OR _sequenceRun = 3 THEN
    IF _sequenceRun = 2 THEN
        _StepIn();
    END_IF

    IF Step(0, TRUE, 'Step 0') THEN
        StepCompleteWhen(TRUE);
    END_IF

    FOR i := 1 TO _totalStepNumber - 2 DO
        Step(i, TRUE, CONCAT('Step ', INT_TO_STRING(i)));
    END_FOR

    IF Step(_totalStepNumber - 1, TRUE, CONCAT('Step ', INT_TO_STRING(_totalStepNumber - 1))) THEN
        CompleteSequence();
    END_IF
END_IF

IF _sequenceRun = 4 THEN
    IF Step(0, TRUE, 'Step 0') THEN
        StepCompleteWhen(TRUE);
    END_IF

    IF Step(1, FALSE, 'Step 1') THEN
        StepCompleteWhen(TRUE);
    END_IF

    FOR i := 2 TO _totalStepNumber - 2 DO
        Step(i, TRUE, CONCAT('Step ', INT_TO_STRING(i)));
    END_FOR

    IF Step(_totalStepNumber - 1, TRUE, CONCAT('Step ', INT_TO_STRING(_totalStepNumber - 1))) THEN
        CompleteSequence();
    END_IF
END_IF

IF _sequenceRun >= 5 THEN
    _StepIn();

    IF Step(0, TRUE, 'Step 0') THEN
        StepCompleteWhen(TRUE);
    END_IF

    IF Step(1, FALSE, 'Step 1') THEN
        StepCompleteWhen(TRUE);
    END_IF

    FOR i := 2 TO _totalStepNumber - 2 DO
        Step(i, TRUE, CONCAT('Step ', INT_TO_STRING(i)));
    END_FOR

    IF Step(_totalStepNumber - 1, TRUE, CONCAT('Step ', INT_TO_STRING(_totalStepNumber - 1))) THEN
        CompleteSequence();
    END_IF
END_IF
END_METHOD

METHOD MAIN_StepModeRequestStepFromHigherToLower
VAR
    i : INT;
END_VAR
IF _sequenceRun <= _reqStep + 5 THEN
    FOR i := 0 TO _reqStep + 4 DO
        _StepIn();

        IF Step(i, TRUE, CONCAT('Step ', INT_TO_STRING(i))) THEN
            StepCompleteWhen(TRUE);
        END_IF
    END_FOR

    FOR i := _reqStep + 5 TO _totalStepNumber - 2 DO
        _StepIn();
        Step(i, TRUE, CONCAT('Step ', INT_TO_STRING(i)));
    END_FOR

    IF Step(_totalStepNumber - 1, TRUE, CONCAT('Step ', INT_TO_STRING(_totalStepNumber - 1))) THEN
        _SequenceComplete();
    END_IF
END_IF

IF _sequenceRun = _reqStep + 6 THEN
    FOR i := 0 TO _reqStep + 4 DO
        _StepIn();

        IF Step(i, TRUE, CONCAT('Step ', INT_TO_STRING(i))) THEN
            StepCompleteWhen(TRUE);
        END_IF
    END_FOR

    FOR i := _reqStep + 5 TO _totalStepNumber - 2 DO
        _StepIn();
        Step(i, TRUE, CONCAT('Step ', INT_TO_STRING(i)));
    END_FOR

    RequestStep(_reqStep);

    IF Step(_totalStepNumber - 1, TRUE, CONCAT('Step ', INT_TO_STRING(_totalStepNumber - 1))) THEN
        _SequenceComplete();
    END_IF
END_IF

IF _sequenceRun >= _reqStep + 7 THEN
    FOR i := 0 TO _totalStepNumber - 1 DO
        _StepIn();
        Step(i, TRUE, CONCAT('Step ', INT_TO_STRING(i)));
    END_FOR

    IF Step(_totalStepNumber, TRUE, CONCAT('Step ', INT_TO_STRING(_totalStepNumber))) THEN
        _SequenceComplete();
    END_IF
END_IF
END_METHOD

METHOD MAIN_StepModeRequestStepFromLowerToHigher
VAR
    i : INT;
END_VAR
IF _sequenceRun = 1 THEN
    IF _currentStep.Status = 20 THEN
        _StepIn();
    END_IF

    IF Step(0, TRUE, 'Step 0') THEN
        StepCompleteWhen(TRUE);
    END_IF

    FOR i := 1 TO _totalStepNumber - 2 DO
        Step(i, TRUE, CONCAT('Step ', INT_TO_STRING(i)));
    END_FOR

    IF Step(_totalStepNumber - 1, TRUE, CONCAT('Step ', INT_TO_STRING(_totalStepNumber - 1))) THEN
        _SequenceComplete();
    END_IF
END_IF

IF _sequenceRun = 2 THEN
    IF _currentStep.Status = 20 THEN
        _StepIn();
    END_IF

    IF Step(0, TRUE, 'Step 0') THEN
        StepCompleteWhen(TRUE);
    END_IF

    RequestStep(_reqStep);

    FOR i := 1 TO _totalStepNumber - 2 DO
        Step(i, TRUE, CONCAT('Step ', INT_TO_STRING(i)));
    END_FOR

    IF Step(_totalStepNumber - 1, TRUE, CONCAT('Step ', INT_TO_STRING(_totalStepNumber - 1))) THEN
        _SequenceComplete();
    END_IF
END_IF
END_METHOD

METHOD MAIN_StepModeStepBackwardFromRunningStep
VAR
    i : INT;
END_VAR
IF _sequenceRun = 1 THEN
    _StepIn();
END_IF

IF _sequenceRun = 11 THEN
    _StepBackward();
END_IF

Step(0, TRUE, 'Step 0');
Step(1, TRUE, 'Step 1');

IF Step(2, TRUE, 'Step 2') THEN
    _StepCompleteWhen(_sequenceRun >= 20);
END_IF

IF Step(3, TRUE, 'Step 3') THEN
    _StepCompleteWhen(_sequenceRun >= 20);
END_IF

FOR i := 4 TO _totalStepNumber - 2 DO
    Step(i, TRUE, CONCAT('Step ', INT_TO_STRING(i)));
END_FOR

IF Step(_totalStepNumber - 1, TRUE, CONCAT('Step ', INT_TO_STRING(_totalStepNumber - 1))) THEN
    CompleteSequence();
END_IF
END_METHOD

METHOD MAIN_StepModeStepForwardBackward
VAR
    i : INT;
END_VAR
IF _sequenceRun = 1 THEN
    FOR i := 0 TO _totalStepNumber - 2 DO
        Step(i, TRUE, CONCAT('Step ', INT_TO_STRING(i)));
    END_FOR

    IF Step(_totalStepNumber - 1, TRUE, CONCAT('Step ', INT_TO_STRING(_totalStepNumber - 1))) THEN
        CompleteSequence();
    END_IF
END_IF

IF _sequenceRun = 2 THEN
    _StepIn();

    IF Step(0, TRUE, 'Step 0') THEN
        StepCompleteWhen(TRUE);
    END_IF

    FOR i := 1 TO _totalStepNumber - 2 DO
        Step(i, TRUE, CONCAT('Step ', INT_TO_STRING(i)));
    END_FOR

    IF Step(_totalStepNumber - 1, TRUE, CONCAT('Step ', INT_TO_STRING(_totalStepNumber - 1))) THEN
        CompleteSequence();
    END_IF
END_IF

IF _sequenceRun = 3 OR _sequenceRun = 5 THEN
    _StepForward();

    IF Step(0, TRUE, 'Step 0') THEN
        StepCompleteWhen(TRUE);
    END_IF

    FOR i := 1 TO _totalStepNumber - 2 DO
        Step(i, TRUE, CONCAT('Step ', INT_TO_STRING(i)));
    END_FOR

    IF Step(_totalStepNumber - 1, TRUE, CONCAT('Step ', INT_TO_STRING(_totalStepNumber - 1))) THEN
        CompleteSequence();
    END_IF
END_IF

IF _sequenceRun = 4 THEN
    RequestStep(_totalStepNumber - 1);

    IF Step(0, TRUE, 'Step 0') THEN
        StepCompleteWhen(TRUE);
    END_IF

    FOR i := 1 TO _totalStepNumber - 2 DO
        Step(i, TRUE, CONCAT('Step ', INT_TO_STRING(i)));
    END_FOR

    IF Step(_totalStepNumber - 1, TRUE, CONCAT('Step ', INT_TO_STRING(_totalStepNumber - 1))) THEN
        CompleteSequence();
    END_IF
END_IF

IF _sequenceRun = 6 OR _sequenceRun = 8 OR _sequenceRun = 9 THEN
    _StepBackward();

    IF Step(0, TRUE, 'Step 0') THEN
        StepCompleteWhen(TRUE);
    END_IF

    FOR i := 1 TO _totalStepNumber - 2 DO
        Step(i, TRUE, CONCAT('Step ', INT_TO_STRING(i)));
    END_FOR

    IF Step(_totalStepNumber - 1, TRUE, CONCAT('Step ', INT_TO_STRING(_totalStepNumber - 1))) THEN
        CompleteSequence();
    END_IF
END_IF

IF _sequenceRun = 7 THEN
    RequestStep(1);

    IF Step(0, TRUE, 'Step 0') THEN
        StepCompleteWhen(TRUE);
    END_IF

    FOR i := 1 TO _totalStepNumber - 2 DO
        Step(i, TRUE, CONCAT('Step ', INT_TO_STRING(i)));
    END_FOR

    IF Step(_totalStepNumber - 1, TRUE, CONCAT('Step ', INT_TO_STRING(_totalStepNumber - 1))) THEN
        CompleteSequence();
    END_IF
END_IF
END_METHOD

METHOD MAIN_StepModeStepForwardFromRunningStep
VAR
    i : INT;
END_VAR
IF _sequenceRun = 1 THEN
    _StepIn();
END_IF

IF _sequenceRun = 11 THEN
    _StepForward();
END_IF

Step(0, TRUE, 'Step 0');
Step(1, TRUE, 'Step 1');

IF Step(2, TRUE, 'Step 2') THEN
    _StepCompleteWhen(_sequenceRun >= 20);
END_IF

IF Step(3, TRUE, 'Step 3') THEN
    _StepCompleteWhen(_sequenceRun >= 20);
END_IF

FOR i := 4 TO _totalStepNumber - 2 DO
    Step(i, TRUE, CONCAT('Step ', INT_TO_STRING(i)));
END_FOR

IF Step(_totalStepNumber - 1, TRUE, CONCAT('Step ', INT_TO_STRING(_totalStepNumber - 1))) THEN
    CompleteSequence();
END_IF
END_METHOD

METHOD MAIN_StepModeStepIn
VAR
    i : INT;
END_VAR
IF _sequenceRun = 1 THEN
    IF Step(0, TRUE, 'Initial step') THEN
        StepCompleteWhen(TRUE);
    END_IF

    FOR i := 1 TO _totalStepNumber - 2 DO
        Step(i, TRUE, CONCAT('Step ', INT_TO_STRING(i)));
    END_FOR

    IF Step(_totalStepNumber - 1, TRUE, CONCAT('Step ', INT_TO_STRING(_totalStepNumber - 1))) THEN
        _SequenceComplete();
    END_IF
END_IF

IF _sequenceRun > 1 THEN
    IF _currentStep.Status = 20 THEN
        _StepIn();
    END_IF

    // Step 0
    IF Step(0, TRUE, 'Step 0') THEN
        StepCompleteWhen(TRUE);
    END_IF

    // Step 1
    IF Step(1, TRUE, 'Step 1') THEN
        StepCompleteWhen(TRUE);
    END_IF

    // Step 2
    IF Step(2, TRUE, 'Step 2') THEN
        StepCompleteWhen(TRUE);
    END_IF

    // Step 3
    IF Step(3, TRUE, 'Step 3') THEN
        StepCompleteWhen(FALSE);
    END_IF

    FOR i := 4 TO _totalStepNumber - 2 DO
        Step(i, TRUE, CONCAT('Step  ', INT_TO_STRING(i)));
    END_FOR

    IF Step(_totalStepNumber - 1, TRUE, CONCAT('Step  ', INT_TO_STRING(_totalStepNumber - 1))) THEN
        _SequenceComplete();
    END_IF
END_IF
END_METHOD

METHOD MAIN_StepModeStepInDetailed
VAR
    i : INT;
END_VAR
IF _sequenceRun = 1 OR _sequenceRun = 5 THEN
    FOR i := 0 TO _totalStepNumber - 2 DO
        Step(i, TRUE, CONCAT('Step ', INT_TO_STRING(i)));
    END_FOR

    IF Step(_totalStepNumber - 1, TRUE, CONCAT('Step ', INT_TO_STRING(_totalStepNumber - 1))) THEN
        CompleteSequence();
    END_IF
END_IF

IF _sequenceRun = 2 THEN
    _StepIn();

    IF Step(0, TRUE, 'Step 0') THEN
        StepCompleteWhen(TRUE);
    END_IF

    FOR i := 1 TO _totalStepNumber - 2 DO
        Step(i, TRUE, CONCAT('Step ', INT_TO_STRING(i)));
    END_FOR

    IF Step(_totalStepNumber - 1, TRUE, CONCAT('Step ', INT_TO_STRING(_totalStepNumber - 1))) THEN
        CompleteSequence();
    END_IF
END_IF

IF _sequenceRun = 3 OR _sequenceRun = 4 THEN
    _StepIn();

    IF Step(0, TRUE, 'Step 0') THEN
        StepCompleteWhen(TRUE);
    END_IF

    IF Step(1, TRUE, 'Step 1') THEN
        RequestStep(_totalStepNumber - 1);
    END_IF

    FOR i := 2 TO _totalStepNumber - 2 DO
        Step(i, TRUE, CONCAT('Step ', INT_TO_STRING(i)));
    END_FOR

    IF Step(_totalStepNumber - 1, TRUE, CONCAT('Step ', INT_TO_STRING(_totalStepNumber - 1))) THEN
        CompleteSequence();
    END_IF
END_IF
END_METHOD

METHOD MAIN_StepModeUncommentPartOfRunningSequencer
VAR
    i : INT;
END_VAR
IF _sequenceRun = 1 THEN
    IF (_currentStep.Status = 20) THEN
        _StepIn();
    END_IF

    IF Step(0, TRUE, 'Step 0') THEN
        StepCompleteWhen(TRUE);
    END_IF

    //	IF Step(1, TRUE, 'Step 1') THEN
    //	   StepCompleteWhen(TRUE);
    //	END_IF
    //	IF Step(2, TRUE, 'Step 2') THEN
    //	   StepCompleteWhen(TRUE);
    //	END_IF
    IF Step(3, TRUE, 'Step 3') THEN
        StepCompleteWhen(FALSE);
    END_IF

    FOR i := 4 TO _totalStepNumber - 2 DO
        IF Step(i, TRUE, CONCAT('Step ', INT_TO_STRING(i))) THEN
            StepCompleteWhen(FALSE);
        END_IF
    END_FOR

    IF Step(_totalStepNumber - 1, TRUE, CONCAT('Step ', INT_TO_STRING(_totalStepNumber - 1))) THEN
        _SequenceComplete();
    END_IF
END_IF

IF _sequenceRun = 2 THEN
    IF (_currentStep.Status = 20) THEN
        _StepIn();
    END_IF

    IF Step(0, TRUE, 'Step 0') THEN
        StepCompleteWhen(TRUE);
    END_IF

    IF Step(1, TRUE, 'Step 1') THEN
        StepCompleteWhen(TRUE);
    END_IF

    IF Step(2, TRUE, 'Step 2') THEN
        StepCompleteWhen(TRUE);
    END_IF

    IF Step(3, TRUE, 'Step 3') THEN
        StepCompleteWhen(FALSE);
    END_IF

    FOR i := 4 TO _totalStepNumber - 2 DO
        IF Step(i, TRUE, CONCAT('Step ', INT_TO_STRING(i))) THEN
            StepCompleteWhen(FALSE);
        END_IF
    END_FOR

    IF Step(_totalStepNumber - 1, TRUE, CONCAT('Step ', INT_TO_STRING(_totalStepNumber - 1))) THEN
        _SequenceComplete();
    END_IF
END_IF
END_METHOD

METHOD MAIN_SwitchStepModeOnDuringStepExecution
VAR
    i : INT;
END_VAR
IF _sequenceRun = 1 THEN
    IF Step(0, TRUE, 'Step 0') THEN
        StepCompleteWhen(TRUE);
    END_IF

    IF Step(1, TRUE, 'Step 1') THEN
        StepCompleteWhen(FALSE);
    END_IF

    FOR i := 2 TO _totalStepNumber - 2 DO
        Step(i, TRUE, CONCAT('Step ', INT_TO_STRING(i)));
    END_FOR

    IF Step(_totalStepNumber - 1, TRUE, CONCAT('Step ', INT_TO_STRING(_totalStepNumber - 1))) THEN
        CompleteSequence();
    END_IF
END_IF

IF _sequenceRun > 1 THEN
    IF Step(0, TRUE, 'Step 0') THEN
        StepCompleteWhen(TRUE);
    END_IF

    IF Step(1, TRUE, 'Step 1') THEN
        IF _sequenceRun >= 5 THEN
            SetStepMode();
        END_IF

        StepCompleteWhen(_sequenceRun >= 10);
    END_IF

    FOR i := 2 TO _totalStepNumber - 2 DO
        Step(i, TRUE, CONCAT('Step ', INT_TO_STRING(i)));
    END_FOR

    IF Step(_totalStepNumber - 1, TRUE, CONCAT('Step ', INT_TO_STRING(_totalStepNumber - 1))) THEN
        CompleteSequence();
    END_IF
END_IF
END_METHOD

METHOD MAIN_SwitchStepModeStepOffFromReadyToRun
VAR
    i : INT;
END_VAR
SetCyclicMode();
Step(0, TRUE, 'Step 0');
Step(1, TRUE, 'Step 1');

IF Step(2, TRUE, 'Step 2') THEN
    _StepCompleteWhen(_sequenceRun >= 20);
END_IF

IF Step(3, TRUE, 'Step 3') THEN
    _StepCompleteWhen(_sequenceRun >= 20);
END_IF

FOR i := 4 TO _totalStepNumber - 2 DO
    Step(i, TRUE, CONCAT('Step ', INT_TO_STRING(i)));
END_FOR

IF Step(_totalStepNumber - 1, TRUE, CONCAT('Step ', INT_TO_STRING(_totalStepNumber - 1))) THEN
    CompleteSequence();
END_IF
END_METHOD

METHOD MAIN_SwitchStepModeStepOffFromRunning
VAR
    i : INT;
END_VAR
SetCyclicMode();
Step(0, TRUE, 'Step 0');
Step(1, TRUE, 'Step 1');

IF Step(2, TRUE, 'Step 2') THEN
    _StepCompleteWhen(_sequenceRun >= 20);
END_IF

IF Step(3, TRUE, 'Step 3') THEN
    _StepCompleteWhen(_sequenceRun >= 20);
END_IF

FOR i := 4 TO _totalStepNumber - 2 DO
    Step(i, TRUE, CONCAT('Step ', INT_TO_STRING(i)));
END_FOR

IF Step(_totalStepNumber - 1, TRUE, CONCAT('Step ', INT_TO_STRING(_totalStepNumber - 1))) THEN
    CompleteSequence();
END_IF
END_METHOD

METHOD MAIN_SwitchStepModeStepOnFromRunning
VAR
    i : INT;
END_VAR
SetStepMode();
Step(0, TRUE, 'Step 0');
Step(1, TRUE, 'Step 1');

IF Step(2, TRUE, 'Step 2') THEN
    _StepCompleteWhen(_sequenceRun >= 20);
END_IF

IF Step(3, TRUE, 'Step 3') THEN
    _StepCompleteWhen(_sequenceRun >= 20);
END_IF

FOR i := 4 TO _totalStepNumber - 2 DO
    Step(i, TRUE, CONCAT('Step ', INT_TO_STRING(i)));
END_FOR

IF Step(_totalStepNumber - 1, TRUE, CONCAT('Step ', INT_TO_STRING(_totalStepNumber - 1))) THEN
    CompleteSequence();
END_IF
END_METHOD

METHOD MAIN_UncommentPartOfRunningSequencer
VAR
    i : INT;
END_VAR
IF _sequenceRun = 1 THEN
    IF Step(0, TRUE, 'Step 0') THEN
        StepCompleteWhen(TRUE);
    END_IF

    //	IF Step(1, TRUE, 'Step 1') THEN
    //	   StepCompleteWhen(TRUE);
    //	END_IF
    //	IF Step(2, TRUE, 'Step 2') THEN
    //	   StepCompleteWhen(TRUE);
    //	END_IF
    IF Step(3, TRUE, 'Step 3') THEN
        StepCompleteWhen(FALSE);
    END_IF

    FOR i := 4 TO _totalStepNumber - 2 DO
        IF Step(i, TRUE, CONCAT('Step ', INT_TO_STRING(i))) THEN
            StepCompleteWhen(FALSE);
        END_IF
    END_FOR

    IF Step(_totalStepNumber - 1, TRUE, CONCAT('Step ', INT_TO_STRING(_totalStepNumber - 1))) THEN
        _SequenceComplete();
    END_IF
END_IF

IF _sequenceRun = 2 THEN
    IF Step(0, TRUE, 'Step 0') THEN
        StepCompleteWhen(TRUE);
    END_IF

    IF Step(1, TRUE, 'Step 1') THEN
        StepCompleteWhen(TRUE);
    END_IF

    IF Step(2, TRUE, 'Step 2') THEN
        StepCompleteWhen(TRUE);
    END_IF

    IF Step(3, TRUE, 'Step 3') THEN
        StepCompleteWhen(FALSE);
    END_IF

    FOR i := 4 TO _totalStepNumber - 2 DO
        IF Step(i, TRUE, CONCAT('Step ', INT_TO_STRING(i))) THEN
            StepCompleteWhen(FALSE);
        END_IF
    END_FOR

    IF Step(_totalStepNumber - 1, TRUE, CONCAT('Step ', INT_TO_STRING(_totalStepNumber - 1))) THEN
        _SequenceComplete();
    END_IF
END_IF
END_METHOD

METHOD PROTECTED OnRestore
_restoreCycleCount := _restoreCycleCount + 1;
END_METHOD

METHOD PROTECTED OnSequenceCompleted
_onSequenceCompleteCount := _onSequenceCompleteCount + 1;
END_METHOD

METHOD PROTECTED OnSequencerError
VAR_INPUT
    inErrorId : eSequencerError;
END_VAR
CASE inErrorId OF
    eSequencerError.noError:
        _onSequencerErrorCount := _onSequencerErrorCount + 0;
    eSequencerError.NotUniqueStepId:
        _onSequencerErrorCount := _onSequencerErrorCount + 10;
    eSequencerError.StepIdHasBeenChanged:
        _onSequencerErrorCount := _onSequencerErrorCount + 20;
    eSequencerError.OrderOfTheStepHasBeenChanged:
        _onSequencerErrorCount := _onSequencerErrorCount + 40;
    eSequencerError.StepWithRequestedIdDoesNotExists:
        _onSequencerErrorCount := _onSequencerErrorCount + 50;
    eSequencerError.MultipleRequestStepMethodCall:
        _onSequencerErrorCount := _onSequencerErrorCount + 60;
    eSequencerError.StepIdTooLow:
        _onSequencerErrorCount := _onSequencerErrorCount + 70;
    eSequencerError.StepIdTooHigh:
        _onSequencerErrorCount := _onSequencerErrorCount + 80;
ELSE
    _onSequencerErrorCount := _onSequencerErrorCount + 0;
END_CASE
END_METHOD

METHOD PROTECTED OnStateChange
VAR_INPUT
    PreviousState : INT;
    NewState : INT;
END_VAR
THIS^._onStateChangeCount := THIS^._onStateChangeCount + 1;
_stateChangeFrom := PreviousState;
_stateChangeTo := NewState;

IF _callRestoreInOnStateChange THEN
    Restore();
END_IF
END_METHOD

METHOD PROTECTED OnStepCompleted
_onCompleteStepCount := _onCompleteStepCount + 1;
END_METHOD

PROPERTY PostOpenRequestStepCycle : UINT
GET
PostOpenRequestStepCycle := _postOpenRequestStepCycle;
END_GET
SET
_postOpenRequestStepCycle := PostOpenRequestStepCycle;
END_SET
END_PROPERTY

PROPERTY PreCloseRequestStepCycle : UINT
GET
PreCloseRequestStepCycle := _preCloseRequestStepCycle;
END_GET
SET
_preCloseRequestStepCycle := PreCloseRequestStepCycle;
END_SET
END_PROPERTY

PROPERTY ReqStep : INT
GET
ReqStep := _reqStep;
END_GET
SET
_reqStep := ReqStep;
END_SET
END_PROPERTY

PROPERTY ReqStepNotExists : INT
GET
ReqStepNotExists := _reqStepNotExists;
END_GET
SET
_reqStepNotExists := ReqStepNotExists;
END_SET
END_PROPERTY

PROPERTY INTERNAL RequestStepCycle : UINT
GET
RequestStepCycle := _requestStepCycle;
END_GET
SET
_requestStepCycle := RequestStepCycle;
END_SET
END_PROPERTY

PROPERTY RunAllSteps : BOOL
GET
RunAllSteps := _runAllSteps;
END_GET
SET
_runAllSteps := RunAllSteps;
END_SET
END_PROPERTY

PROPERTY RunOneStep : BOOL
GET
RunOneStep := _runOneStep;
END_GET
SET
_runOneStep := RunOneStep;
END_SET
END_PROPERTY

{attribute 'TcRpcEnable'}
METHOD SaveNumberOfStepsInSequence
_numberOfSteps := THIS^._numberOfStepsInSequence;
_previousNumberOfSteps := THIS^._previousNumberOfStepsInSequence;
END_METHOD

PROPERTY SequenceCycles : UINT
GET
SequenceCycles := _sequenceCycles;
END_GET
SET
_sequenceCycles := SequenceCycles;
END_SET
END_PROPERTY

METHOD INTERNAL SequencerClose
SUPER^._Close();
END_METHOD

METHOD INTERNAL SequencerOpen
SUPER^._Open();
END_METHOD

PROPERTY SequenceRun : ULINT
GET
SequenceRun := _sequenceRun;
END_GET
SET
_sequenceRun := SequenceRun;
END_SET
END_PROPERTY

{attribute 'TcRpcEnable'}
METHOD INTERNAL SetChildState
VAR_INPUT
    inState : INT;
END_VAR
THIS^._myTcoChildState.ChangeState(inState);
END_METHOD

{attribute 'TcRpcEnable'}
METHOD INTERNAL SetCurrentStep
VAR_INPUT
    inStepID : INT;
    inStepDescription : STRING(254);
END_VAR
THIS^._currentStep.ID := inStepID;
THIS^._currentStep.Description := inStepDescription;
END_METHOD

{attribute 'TcRpcEnable'}
METHOD SetCurrentStepToErrorState : BOOL
_currentStep.Status := TcoCore.eStepStatus.Error;
SetCurrentStepToErrorState := _currentStep.Status = TcoCore.eStepStatus.Error;
END_METHOD

METHOD SetCyclicMode : BOOL
ModeController.Mode := eSequencerMode.CyclicMode;
SetCyclicMode := ModeController.Mode = eSequencerMode.CyclicMode;
END_METHOD

{attribute 'TcRpcEnable'}
METHOD SetInvalidMode : BOOL
ModeController.Mode := eSequencerMode.Invalid;
SetInvalidMode := ModeController.Mode = eSequencerMode.Invalid;
END_METHOD

METHOD INTERNAL SetNumberOfSteps
VAR_INPUT
    inNumberOfSteps : UINT;
END_VAR
_stepCounter := inNumberOfSteps;
_numberOfStepsInSequence := inNumberOfSteps;
_previousNumberOfStepsInSequence := inNumberOfSteps;
END_METHOD

METHOD INTERNAL SetSequenceAsChecked
_stepIDUniquenessChecked := TRUE;
_StepIdUniquenessControlState := eStepIdUniquenessControlState.Done;
END_METHOD

METHOD INTERNAL SetSequenceAsNotChecked
_stepIDUniquenessChecked := FALSE;
_StepIdUniquenessControlState := eStepIdUniquenessControlState.NotYetStarted;
END_METHOD

METHOD SetStepMode : BOOL
ModeController.Mode := eSequencerMode.StepMode;
SetStepMode := ModeController.Mode = eSequencerMode.StepMode;
END_METHOD

{attribute 'TcRpcEnable'}
METHOD INTERNAL SetupChildRequestedState
VAR_INPUT
    inState : INT;
END_VAR
THIS^._myTcoChildState.RequestedState := inState;
END_METHOD

PROPERTY StepDescription : STRING(254);
GET
StepDescription := _stepDescription;
END_GET
SET
_stepDescription := StepDescription;
END_SET
END_PROPERTY

PROPERTY StepId : INT
GET
StepId := _stepId;
END_GET
SET
_stepId := StepId;
END_SET
END_PROPERTY

PROPERTY StepInEvents : UINT
GET
StepInEvents := _stepInEvents;
END_GET
SET
_stepInEvents := StepInEvents;
END_SET
END_PROPERTY

PROPERTY TcoSequencerTest : eTcoSequenceTests
GET
TcoSequencerTest := _tcoSequenceTest;
END_GET
SET
_tcoSequenceTest := TcoSequencerTest;
END_SET
END_PROPERTY

PROPERTY TotalStepNumber : UINT
GET
TotalStepNumber := _totalStepNumber;
END_GET
SET
_totalStepNumber := TotalStepNumber;
END_SET
END_PROPERTY

END_FUNCTION_BLOCK

(* stored: Version 1.1.0.1
   POU TcoSequenceTestType: Id {a078dca2-adb3-097e-327d-7525ae7a7cb8}, SpecialFunc None
   Folder _Tests: Id {b2693abd-bbc8-0e03-2dee-8c9184f59647}
   Folder MAINS: Id {e0f15297-fee6-07d1-2f94-d23d4c9b552c}
   Method _RequestStep: Id {c95b942f-a2c0-0823-1832-45c1d2992fd2}
   Method _RunExecutionSubstitute: Id {f008b1d2-34fa-092d-16be-28669f572893}
   Method _SequenceComplete: Id {0d07da38-add0-0d55-108f-09e3b9860458}
   Method _Step: Id {083d38ba-2338-03c7-3e04-25519c175d87}
   Method _StepBackward: Id {ce086e2c-ea79-0ad3-16db-f3609abcd4b3}
   Method _StepCompleteWhen: Id {1cd51cd6-1ec5-03ab-0b25-98134af6df4e}
   Method _StepForward: Id {601c61da-43de-058c-178b-70930ce2cb8d}
   Method _StepIn: Id {cd8c3752-6fef-0e86-2668-fe4727637839}
   Property CallRestoreInOnStateChange: Id {a1f545f7-c7d5-0cbc-039e-8b4e2c38ecee}
   Get Get: Id {c7824f5b-c573-069d-1aab-e1c6618ddd6b}
   Set Set: Id {8eb6e2c7-e5df-052c-286b-c87c7968dba3}
   Method ChildHasAutoRestoreEnabled: Id {da4e96fa-8b8f-0db8-1b1a-b964d6f92f79}
   Method ChildIsAutoRestorable: Id {dd6980f6-e7a2-003d-3677-6c6447bc161e}
   Method ClearNumberOfSteps: Id {26c5d13b-8880-0206-09f0-db807701b452}
   Property CyclicCycles: Id {b6f5d22a-fc3e-0716-3271-b4eea83f4200}
   Get Get: Id {fe9b89cc-acea-02aa-2ad8-16be016a0875}
   Set Set: Id {b2e2610a-5d08-05f0-30ed-6dde0ffc46d4}
   Property Enabled: Id {1087fd9d-eb9e-0e13-19aa-b3081e9d0f29}
   Get Get: Id {d2454bf6-abef-0c51-0fb7-175a8e7cc33b}
   Set Set: Id {f5c67497-5008-028a-1cb0-a4c1ce649695}
   Property FinishStep: Id {7dd360d5-d280-0c9a-2b7e-2bbacf96ec70}
   Get Get: Id {b4922eaa-b2df-031a-0c5c-52991636c289}
   Set Set: Id {ef720c61-781e-0c73-0c29-599f59a3b545}
   Method GetChildState: Id {3c61e758-881e-07ce-2657-5146ba932ce9}
   Method GetOrderOfTheCurrentlyEvaluatedStep: Id {312eb82a-831e-0196-3a25-d23bd8aef8c8}
   Method GetOrderOfTheCurrentlyExecutedStep: Id {267f659b-caa9-02f8-2e8e-b9bacf7af60c}
   Method GetRequestStepCycle: Id {62ed0e0f-86de-050e-0799-aef70f8e4bcf}
   Method HasAutoRestoreEnabled: Id {66fbc43c-5014-017c-3394-28486ed441e5}
   Property InitReqStepCycle: Id {2884ff71-7bb3-071f-37a9-de1b2d25ae11}
   Get Get: Id {2643949e-2357-0299-0594-754926cdf200}
   Set Set: Id {57b53abf-69b2-0f0d-1dad-69c7b8c2c237}
   Method IsAutoRestorable: Id {e3b93f74-745d-08cd-331a-375a0d45cebb}
   Method Main: Id {7cd483d4-4c79-0cb8-3ef2-900b7113f4aa}
   Method MAIN_ChangeStepIdDuringExecution: Id {c3e35577-8969-0f7a-25fc-2d3e2211a756}
   Method MAIN_CheckStepIdUniqueness: Id {94d68c00-42c5-06e5-19fb-7b168034f84b}
   Method MAIN_CommentOutPartOfRunningSequencer: Id {71fa6f12-9cd1-0764-19c7-65883cf277d1}
   Method MAIN_ExecutionInOnePLCcycle: Id {df3fc404-c332-0991-0741-c71c254c84bf}
   Method MAIN_MaxStepId: Id {6e483f01-ba14-0f16-1bc7-8c0dc743b277}
   Method MAIN_MinStepId: Id {a62d3e76-a8e0-0f2e-12d9-99c6ca676bac}
   Method MAIN_NumberOfStepsCount: Id {24259989-41e3-0d4c-3980-d3f83add522d}
   Method MAIN_OnStateChangeWhenChangingModes: Id {66b3a3ec-ed4f-0536-304f-3abf886c8bec}
   Method MAIN_RequestStep: Id {198ed2c1-0d74-0033-03b4-f7268587ca06}
   Method MAIN_RequestStepFromHigherToLower: Id {173d6e19-ec12-09f3-3657-552bbf2ee8ff}
   Method MAIN_RequestStepFromLowerToHigher: Id {ac379fce-6f90-076f-0f33-f781c47fc5bf}
   Method MAIN_RequestStepToFirstStepWithStepId0: Id {3c1e2b30-a8d1-0876-3543-45f8a1ef6bd7}
   Method MAIN_RequestStepToNotExistingStep: Id {9f2d0e9b-5ee0-0444-3ac8-b2acf625df04}
   Method MAIN_RequestStepWhilePreviousRequestStepHasNotBeenYetProcessed: Id {13885226-cac1-0bac-0919-fa6ea31c8772}
   Method MAIN_RestoreChildBetweenSteps: Id {bc467ad1-9715-0d90-255c-9c7e93d80d14}
   Method MAIN_SetStepMode: Id {c8954608-0f9b-0e60-2965-44cc8609a07d}
   Method MAIN_StepMode: Id {55a75494-51cd-061d-2d8b-31e4481e05f2}
   Method MAIN_StepModeChangeStepIdDuringExecution: Id {1116d3f0-e241-07b4-1956-abe49a29fcdf}
   Method MAIN_StepModeChangeStepOrder: Id {41237a48-2c9b-0a10-2b82-277c049a95e8}
   Method MAIN_StepModeCommentOutPartOfRunningSequencer: Id {100634a5-64cb-093d-00f1-41c535fdc4eb}
   Method MAIN_StepModeDisabledStep: Id {f314ae6d-ba2a-0c87-2c0f-932cf34b4ce5}
   Method MAIN_StepModeRequestStepFromHigherToLower: Id {2a14da23-88e1-0e24-1ec4-ecf46bfd64ac}
   Method MAIN_StepModeRequestStepFromLowerToHigher: Id {ce362780-51b7-07a7-1cf8-36c6219376f5}
   Method MAIN_StepModeStepBackwardFromRunningStep: Id {739c3154-4164-0849-2911-133282de98e4}
   Method MAIN_StepModeStepForwardBackward: Id {2c7298e9-ddc6-054c-09e1-7d092809dffe}
   Method MAIN_StepModeStepForwardFromRunningStep: Id {61b23bc4-218a-0e07-052d-5c69743369a7}
   Method MAIN_StepModeStepIn: Id {e5736456-11e0-01df-1d83-672610ff8007}
   Method MAIN_StepModeStepInDetailed: Id {df946c0e-e1f0-08b2-31fd-00db6d6f556d}
   Method MAIN_StepModeUncommentPartOfRunningSequencer: Id {fa6ef621-d917-0fa9-18d8-34b8354d15b1}
   Method MAIN_SwitchStepModeOnDuringStepExecution: Id {16c90f55-993d-0561-35eb-a0aeb9d3db7a}
   Method MAIN_SwitchStepModeStepOffFromReadyToRun: Id {32a7c0a6-2180-0554-2f60-a1ada697be68}
   Method MAIN_SwitchStepModeStepOffFromRunning: Id {001d6e24-4c3a-0c64-24a6-61067704836e}
   Method MAIN_SwitchStepModeStepOnFromRunning: Id {2b458c99-1b1a-0bf6-1afa-6a09733b094a}
   Method MAIN_UncommentPartOfRunningSequencer: Id {49646959-6e36-01e8-260c-1f55f5ec7fc9}
   Method OnRestore: Id {f1c046c4-e6d7-0fa8-39c8-970edc9f12be}
   Method OnSequenceCompleted: Id {60298763-4824-09b1-2830-be21d8dcaa4e}
   Method OnSequencerError: Id {fb11aee0-1df3-0d7f-03b6-1d9211fb2b0f}
   Method OnStateChange: Id {e9815ab8-29e5-062b-1852-98a159765651}
   Method OnStepCompleted: Id {ddd486f4-6c54-07e5-3977-6d0473cb44b6}
   Property PostOpenRequestStepCycle: Id {3be1f7f2-d985-03fa-0786-a8933695867e}
   Get Get: Id {7472050e-4120-0a24-1f18-8f6e6bb926ab}
   Set Set: Id {8a6e010a-6d7d-09f2-0286-1fe833bc7501}
   Property PreCloseRequestStepCycle: Id {302b02a6-ec70-0aa6-115e-3d7d15f8d0f0}
   Get Get: Id {557a7b98-0f87-0e98-0405-360da897ca44}
   Set Set: Id {cae3c77d-c393-02d2-0365-bd0ee616af4b}
   Property ReqStep: Id {7dbede49-78a4-0c54-332d-b479f564d0de}
   Get Get: Id {ccb030b6-b8a0-070f-1bb2-4b4f1fe7a1f7}
   Set Set: Id {ef57e2c3-34c9-00f6-1646-753997a02fb9}
   Property ReqStepNotExists: Id {7b130003-26d4-0204-38e2-f876d2a22bbb}
   Get Get: Id {89e91174-8037-0619-3841-36b7a23c8b87}
   Set Set: Id {38a8284e-8fc3-07dc-0a90-9fdbd889b646}
   Property RequestStepCycle: Id {bda0e552-817a-067e-0895-613878e0f39a}
   Get Get: Id {02fb61fa-4cd8-0b30-22bf-f6a1251a7177}
   Set Set: Id {213dbda0-686d-0774-1866-56f8d78559af}
   Property RunAllSteps: Id {87216f2b-5006-05c9-2d80-73c5a95853aa}
   Get Get: Id {956e824f-8661-065c-0374-08ff2779aa2c}
   Set Set: Id {e7862909-659e-0b9b-15cc-1cdcfa8fa5c8}
   Property RunOneStep: Id {67ef8b0a-90a9-0880-10de-5f05032f8a06}
   Get Get: Id {8d6d89ad-7dac-0670-3219-15320ad6aeea}
   Set Set: Id {5dbe4c02-1be9-059c-2d10-3f282212a60b}
   Method SaveNumberOfStepsInSequence: Id {bf56cbc7-5304-07bb-0341-b1d009e5e5ac}
   Property SequenceCycles: Id {0dc7b43b-5dd7-03f4-1814-0911e8b39393}
   Get Get: Id {8f7689aa-b65c-08aa-3a07-2e66f65c6844}
   Set Set: Id {c59ae70b-eafe-09f9-0a89-c64bc887cc9e}
   Method SequencerClose: Id {5cccc8f6-8740-0c81-3163-241e13fcbeb6}
   Method SequencerOpen: Id {31aab523-a57b-028e-1000-2e46dbf7483b}
   Property SequenceRun: Id {d6112955-355b-0178-3ba4-bb2f212985f4}
   Get Get: Id {bbb199c9-f2b8-0c73-1d68-9cf1db227751}
   Set Set: Id {7389e3b2-b6a4-002e-3417-721dac6d658b}
   Method SetChildState: Id {ca54244a-6d31-0632-05fb-fb3e6fa5d119}
   Method SetCurrentStep: Id {f17f581f-7d98-0644-0c00-f263d0dfa946}
   Method SetCurrentStepToErrorState: Id {210f6dc4-adf4-0e2b-3e75-6cbd34cf51e4}
   Method SetCyclicMode: Id {bfbf5225-839d-0c49-021c-5ca0db52c603}
   Method SetInvalidMode: Id {5ddc53f7-d2c6-0855-0a9c-e60a2b64947f}
   Method SetNumberOfSteps: Id {f8d0f7aa-093e-0131-12ce-c1fa912c1d32}
   Method SetSequenceAsChecked: Id {4326a977-738e-0b21-3421-c92a826986ad}
   Method SetSequenceAsNotChecked: Id {0e043be6-f20b-0526-1c74-dadaf5fede50}
   Method SetStepMode: Id {6c94eaba-bcb8-0e97-34d9-b3ee7c3ee17e}
   Method SetupChildRequestedState: Id {5a5235ff-1915-0a32-2b03-9bcc9425c4d0}
   Property StepDescription: Id {7dc35663-a4b9-0a1b-083b-d7ec981d8b48}
   Get Get: Id {24687b75-d257-0c86-0fbc-c080703770d4}
   Set Set: Id {6c55d23c-d64e-04ff-20f2-85228c761936}
   Property StepId: Id {08c4baf8-c0bb-0bda-2595-c00c37aea189}
   Get Get: Id {2357a271-d5c9-0ddd-1136-3ca5f7b3b17c}
   Set Set: Id {7121188d-d908-0fc9-3da3-1f10d83400dc}
   Property StepInEvents: Id {79db699c-e247-0a5e-070e-070be1abe34d}
   Get Get: Id {ec5bca7c-67e5-0f65-26e7-a9bf85c33073}
   Set Set: Id {07f03407-70b4-08db-149e-6a1337fa3ddd}
   Property TcoSequencerTest: Id {00bd0fac-3ac4-0048-19e4-759610100930}
   Get Get: Id {cde7a63e-f575-0470-307f-5600c34f9837}
   Set Set: Id {6db9ec71-8905-0610-1059-e92e549ed779}
   Property TotalStepNumber: Id {511cc388-c125-0ad8-0046-6f0984089ec4}
   Get Get: Id {e5be93c8-9592-0b7d-2029-35c59093f619}
   Set Set: Id {8bcdbd8b-921f-0cd3-1e4a-1e93d6981e36} *)
